// TwinCAT 3 PLC project TcOtel
// Title: TcOtel
// Company: AVM Engineering
// Author: Pirmin Bleiker
// ProjectVersion: 0.0.1
// ProgramVersion: 3.1.4026.22
// CompilerDefines: DEBUG
// libraries:
//   Tc2_EtherCAT, * (Beckhoff Automation GmbH)
//   Tc2_Standard, * (Beckhoff Automation GmbH)
//   Tc2_System, * (Beckhoff Automation GmbH)
//   Tc2_Utilities, * (Beckhoff Automation GmbH)
//   Tc3_Module, * (Beckhoff Automation GmbH)
//   TcUnit, * (www.tcunit.org)
//   Base Interfaces,newest,System
// project tree:
//   API/Context/ FB_ScopedContext.TcPOU, F_Context.TcPOU, I_ContextBuilder.TcIO
//   API/Log/ E_LogLevel.TcDUT, FB_Log.TcPOU (not stored), F_Log.TcPOU
//   API/Metric/ E_MetricStat.TcDUT, FB_Metrics.TcPOU
//   API/Trace/ FB_Trace.TcPOU (not stored), FB_Span.TcPOU (not stored), F_TraceParentFromString.TcPOU
//   API/Log/Interface/ I_LogBuilder.TcIO, I_WithLogger.TcIO, I_WithContext.TcIO, I_Logger.TcIO
//   API/ PRG_TaskLog.TcPOU (not stored)
//   DUTs/ E_CustomTypes.TcDUT, E_Scope.TcDUT, ST_TcOtelTaskInfo.TcDUT, ST_ScopedContextStack.TcDUT, E_TypeIdV2.TcDUT, ST_LogEntryHeaderV2.TcDUT, ST_SpanBeginPrefix.TcDUT, ST_SpanAttrFrame.TcDUT, ST_SpanEventFrame.TcDUT, ST_SpanEndFrame.TcDUT
//   GVLs/ Config.TcGVL (not stored), Const.TcGVL, TcOtelInfo.TcGVL
//   ITFs/ I_LogEntry.TcIO, I_LogEntryAdder.TcIO
//   POUs/Diagnostic/ FB_TcOtelTaskDiag.TcPOU, ST_PushDiagBatchHeader.TcDUT, ST_PushDiagConfig.TcDUT, ST_PushDiagSample.TcDUT
//   POUs/Logs/ FB_ContextBuilder.TcPOU, FB_LogBuilder.TcPOU, FB_LogEntry.TcPOU
//   POUs/Metrics/ E_MetricBodySchema.TcDUT, FB_TcOtelTaskMetrics.TcPOU, ST_DiagnosticCalculations.TcDUT, ST_PushMetricAggHeader.TcDUT
//   POUs/Trace/ E_SpanKind.TcDUT, E_SpanStatus.TcDUT, F_HashSpanId.TcPOU, F_HashTraceId.TcPOU, FB_TcOtelTaskTracer.TcPOU (not stored)
//   POUs/ FB_TcOtelTask.TcPOU (not stored), F_InternalLog.TcPOU (not stored), PRG_ScopedContextStack.TcPOU
//   POUs/Utils/ FB_LogBuffer.TcPOU, F_DINT_TO_UINT_MAX.TcPOU, IncUDINT.TcPOU
//   / ApiTest.TcPOU
//   Test/ FB_ContextBuilder_Test.TcPOU, PlcTask.TcTTO, PRG_Test.TcPOU
//   Version/ Global_Version.TcGVL
// real-time tasks:
//   TASK PlcTask: cycle T#1ms, priority 20, ADS port 350

CONFIGURATION TcOtel
    RESOURCE PLC ON TwinCAT3
        TASK PlcTask(INTERVAL := T#1ms, PRIORITY := 20);
        PROGRAM PRG_Test WITH PlcTask : PRG_Test;
    END_RESOURCE
END_CONFIGURATION

// ---- API/Log/E_LogLevel.TcDUT
(*
:Description: Definition of available log levels. 

The log levels are ordered. ``eTrace`` has the lowest priority, ``eFatal`` has the
highest priority.

===============
Log Level Usage
===============

Is is recommended to build a guidline for consistent use of the log level. A example
could be the following:

:eFatal: The fatal level should be used for any error which will to malfunction of the most
	part of the program. Log message of this type must be handled immedialtely.
	
	Example: A Safety controller could not be initialised

:eError: The error level should be used when the program cannot continue to work properly.
	Normally this means that a operator/user has to be alerted and something has to
	be fixed.

	Example: Communication errors, something stops a process

:eWarn: The warn level should be used when some expected condition has happend, but the
	software can proceed in some way or the operation can be repeated later. Normaly
	the warn level should be read by the user/operator at some time, not necessarly 
	immediately.

	Example: Cannot connect to some external system (but will repeat to try)

:eInfo: The info level should track some of the import state changes in the programm. This
	information can be used by the user/operator on demand to track a problem.

	Example: A state of a state-machine has changed, a new recipe has been loaded

:eDebug: The info level should track of the some internals, normally only of importance to
	developers.

:eTrace: The trace level should be used to track some internal processing. This is rarely
	used, even by developers, mostly to track some difficult problem.

*)
{attribute 'qualified_only'}
{attribute 'strict'}
{attribute 'to_string'}
TYPE E_LogLevel :
(
	eTrace 	:= 0,	(* Trace log level. *)
	eDebug 	:= 1,	(* Debug log level. *)
	eInfo	:= 2,	(* Info log level. *)
	eWarn	:= 3,	(* Warn log level. *)
	eError	:= 4,	(* Error log level. *)
	eFatal	:= 5,	(* Fatal log level. *)
	eDisabled := 99	(* Disabled *)
) UINT;
END_TYPE

// ---- API/Metric/E_MetricStat.TcDUT
(*
:Description: Bitmask values for the FB_Metrics aggregation stats.

Each bit selects one statistic that will be computed online (Welford
algorithm for mean / variance) over each sample interval and shipped as
8 bytes inside the body of an FB_Metrics aggregate frame
(``body_schema = eNumericAggregated``).

The wire-side ``nStatMask`` byte at header offset +0x11 is the OR of
the selected values. Body sample size = ``popcount(mask) * 8``. Stats
are written into the body in **bit-index order** (Min first if set,
then Max, then Mean, then Sum, then Count, then StdDev) — the decoder
walks the mask bit-by-bit and reads 8 bytes per set bit.

OR the values together to pick the stats you want:

.. code-block:: pascal

    fb.SetAggregation(E_MetricStat.eSum);                                   // counter
    fb.SetAggregation(E_MetricStat.eMin OR E_MetricStat.eMax);              // envelope
    fb.SetAggregation(E_MetricStat.eMin OR E_MetricStat.eMax
                      OR E_MetricStat.eMean);                               // recommended
    fb.SetAggregation(E_MetricStat.eMin OR E_MetricStat.eMax
                      OR E_MetricStat.eMean OR E_MetricStat.eSum
                      OR E_MetricStat.eCount OR E_MetricStat.eStdDev);      // full

Single-stat selections are valid and useful — e.g. ``eSum`` alone for
energy / counter metrics.
*)
TYPE E_MetricStat :
(
    eMin    := 16#01,    // bit 0
    eMax    := 16#02,    // bit 1
    eMean   := 16#04,    // bit 2 — Welford online mean
    eSum    := 16#08,    // bit 3 — total over the sample interval
    eCount  := 16#10,    // bit 4 — number of Observe() calls aggregated
    eStdDev := 16#20     // bit 5 — Welford online sample stddev
) BYTE;
END_TYPE

// ---- DUTs/E_CustomTypes.TcDUT
{attribute 'pack_mode' := '1'}
{attribute 'qualified_only'}
{attribute 'strict'}
TYPE INTERNAL E_CustomTypes :
(
	eType_TIME				:= 20000,
	eType_LTIME				:= 20001,
	eType_DATE				:= 20002,
	eType_DATE_AND_TIME		:= 20003,
	eType_TIME_OF_DAY		:= 20004,
	eType_ENUM				:= 20005,
	eType_WSTRING			:= 20006
) INT;
END_TYPE

// ---- DUTs/E_Scope.TcDUT
{attribute 'pack_mode' := '1'}
{attribute 'qualified_only'}
{attribute 'strict'}
{attribute 'conditionalshow'}
{attribute 'to_string'}
TYPE E_Scope :
(
	eLog			:= 0,
	eLogger			:= 1,
	eScoped			:= 2,
	eTask			:= 3
) BYTE;
END_TYPE

// ---- DUTs/ST_TcOtelTaskInfo.TcDUT
TYPE ST_TcOtelTaskInfo :
STRUCT
	nAddLogToBuffer						: UDINT;	(* Counts number of logs added to message buffer. *)
	nAddLogToBufferErrorCount			: UDINT;	(* Counts error when adding log message to task buffer. *)
	nSendLogBufferErrorCount			: UDINT;	(* Counts error when sending log task buffer to service. *)
	nMaxUsedBufferSize					: UDINT;	(* Max. used buffer size of log task buffer. *)
	bConnected							: BOOL;		(* TRUE when the service is reachable (last send succeeded). Logs are suppressed while FALSE. *)
	bReconnectPending					: BOOL;		(* TRUE on FALSE->TRUE bConnected edge; consumed by the task to emit a one-shot reconnect log. *)
END_STRUCT
END_TYPE

// ---- DUTs/ST_ScopedContextStack.TcDUT
{attribute 'conditionalshow'}
TYPE INTERNAL ST_ScopedContextStack :
STRUCT
	aScopedContext		: ARRAY[0..Config.nMaxScopedContext-1] OF I_ContextBuilder;
	nScopeContextCount	: UINT (0..Config.nMaxScopedContext);
END_STRUCT
END_TYPE

// ---- DUTs/E_TypeIdV2.TcDUT
{attribute 'pack_mode' := '1'}
{attribute 'qualified_only'}
{attribute 'strict'}
TYPE INTERNAL E_TypeIdV2 :
(
	eType_TIME_V2			:= 100,
	eType_LTIME_V2			:= 101,
	eType_DATE_V2			:= 102,
	eType_DATE_AND_TIME_V2	:= 103,
	eType_TIME_OF_DAY_V2	:= 104,
	eType_ENUM_V2			:= 105,
	eType_WSTRING_V2		:= 106
) BYTE;
END_TYPE

// ---- DUTs/ST_LogEntryHeaderV2.TcDUT
{attribute 'pack_mode' := '1'}
TYPE INTERNAL ST_LogEntryHeaderV2 :
STRUCT
	nType			: BYTE;		// 0x02 for v2 log entry
	nEntryLength	: UINT;		// Total length from after this field
	nLevel			: BYTE;		// Log level
	nTsPlc			: LINT;		// PLC timestamp (FILETIME)
	nTsClock		: LINT;		// Clock timestamp (FILETIME)
	nTaskIndex		: BYTE;		// Task index (0-63)
	nCycleCount		: UDINT;	// Cycle counter
	nArgCount		: BYTE;		// Argument count
	nContextCount	: BYTE;		// Context group count
END_STRUCT
END_TYPE

// ---- DUTs/ST_SpanBeginPrefix.TcDUT
(*
Fixed 24-byte prefix of a SPAN_BEGIN frame. Trace_id (16B) and span_id (8B)
follow immediately after, then the variable-length name and optional
external traceparent. Layout matches Rust parser_v2 BEGIN case.
*)
{attribute 'pack_mode' := '1'}
TYPE INTERNAL ST_SpanBeginPrefix :
STRUCT
    (* 12-byte common header *)
    nEventType      : BYTE;     (* 5 = SPAN_BEGIN *)
    nLocalId        : BYTE;     (* monotonic counter for SpanKey uniqueness *)
    nTaskIdx        : BYTE;
    nFlags          : BYTE;     (* bit1 = has_external_parent *)
    nDcTime         : LINT;     (* ns since DC epoch *)
    (* 12-byte begin meta *)
    abParentSpanId  : ARRAY[0..7] OF BYTE;
    nKind           : BYTE;
    nNameLen        : BYTE;
    nReserved       : ARRAY[0..1] OF BYTE;
END_STRUCT
END_TYPE

// ---- DUTs/ST_SpanAttrFrame.TcDUT
(*
Fixed 23-byte header of a SPAN_ATTR frame. Followed by key (nKeyLen bytes)
and value (nValueLen bytes). Layout matches Rust parser_v2 ATTR case.
*)
{attribute 'pack_mode' := '1'}
TYPE INTERNAL ST_SpanAttrFrame :
STRUCT
    (* 12-byte common header *)
    nEventType      : BYTE;     (* 6 = SPAN_ATTR *)
    nSpanIdByte0    : BYTE;     (* span_id[0] — shares slot with local_id *)
    nTaskIdx        : BYTE;
    nFlags          : BYTE;
    nDcTime         : LINT;
    (* 7-byte span_id rest *)
    abSpanIdRest    : ARRAY[0..6] OF BYTE;
    (* 4-byte attr meta *)
    nValueType      : BYTE;     (* 1=i64, 2=f64, 3=bool, 4=string *)
    nKeyLen         : BYTE;     (* ≤31 *)
    nValueLen       : BYTE;     (* wire bytes for value (1/8/N) *)
    nReserved       : BYTE;
END_STRUCT
END_TYPE

// ---- DUTs/ST_SpanEventFrame.TcDUT
(*
Fixed 23-byte header of a SPAN_EVENT frame. Followed by name (nNameLen bytes).
Layout matches Rust parser_v2 EVENT case.
*)
{attribute 'pack_mode' := '1'}
TYPE INTERNAL ST_SpanEventFrame :
STRUCT
    nEventType      : BYTE;     (* 7 = SPAN_EVENT *)
    nSpanIdByte0    : BYTE;
    nTaskIdx        : BYTE;
    nFlags          : BYTE;
    nDcTime         : LINT;
    abSpanIdRest    : ARRAY[0..6] OF BYTE;
    nNameLen        : BYTE;     (* ≤31 *)
    nAttrCount      : BYTE;     (* always 0 — inline attrs unused *)
    nReserved       : ARRAY[0..1] OF BYTE;
END_STRUCT
END_TYPE

// ---- DUTs/ST_SpanEndFrame.TcDUT
(*
Fixed 23-byte SPAN_END frame — no variable payload.
Layout matches Rust parser_v2 END case.
*)
{attribute 'pack_mode' := '1'}
TYPE INTERNAL ST_SpanEndFrame :
STRUCT
    nEventType      : BYTE;     (* 8 = SPAN_END *)
    nSpanIdByte0    : BYTE;
    nTaskIdx        : BYTE;
    nFlags          : BYTE;
    nDcTime         : LINT;
    abSpanIdRest    : ARRAY[0..6] OF BYTE;
    nStatus         : BYTE;     (* 1 = ok, 2 = error *)
    nMsgLen         : BYTE;     (* 0 — status_msg unused on wire today *)
    nReserved       : ARRAY[0..1] OF BYTE;
END_STRUCT
END_TYPE

// ---- POUs/Diagnostic/ST_PushDiagBatchHeader.TcDUT
(*
:Description: 80-byte header of a per-task diagnostic batch frame.

Prepended to an array of ``ST_PushDiagSample`` entries before pushing via
``ADSWRITE`` to tc-otel (IG = 16#4D424301, IO = 0). Packed tight
(``pack_mode := 1``) so on-wire layout matches the decoder in tc-otel-ads.
*)
  {attribute 'pack_mode' := '1'}
TYPE INTERNAL ST_PushDiagBatchHeader :
STRUCT
  version            : BYTE;                        // +0x00, wire version = 2
  event_type         : BYTE;                        // +0x01, event_type = 10 (batch)
  reserved0          : UINT;                        // +0x02, reserved = 0
  task_obj_id        : UDINT;                       // +0x04, TwinCAT task object id
  task_port          : UINT;                        // +0x08, AMS port of the owning task
  window_ms          : UINT;                        // +0x0A, aggregation window used for this batch (ms)
  sample_count       : UINT;                        // +0x0C, number of ST_PushDiagSample entries following
  reserved1          : UINT;                        // +0x0E, reserved = 0
  cycle_count_start  : UDINT;                       // +0x10, task cycle counter at first sample
  cycle_count_end    : UDINT;                       // +0x14, task cycle counter at last sample
  dc_time_start      : LINT;                        // +0x18, DC time at first sample (ns)
  dc_time_end        : LINT;                        // +0x20, DC time at last sample (ns)
  exec_time_min_us   : UDINT;                       // +0x28, min exec time in window (us)
  exec_time_max_us   : UDINT;                       // +0x2C, max exec time in window (us)
  exec_time_avg_us   : UDINT;                       // +0x30, avg exec time in window (us)
  cycle_exceed_count : UDINT;                       // +0x34, exceed cycles in window
  rt_violation_count : UDINT;                       // +0x38, rt-violation cycles in window
  task_name          : ARRAY [0..19] OF BYTE;       // +0x3C, task name (null-padded)
END_STRUCT
END_TYPE

// ---- POUs/Diagnostic/ST_PushDiagConfig.TcDUT
(*
:Description: Per-task push-diagnostic configuration, writable from tc-otel.

One instance per task lives in ``PRG_TaskLog.aTaskDiagConfig``. tc-otel can
update these slots at runtime via ADS SymbolByName writes so operators can
tune the aggregation window or disable push diagnostics from the UI without
recompiling the PLC project.

``divider = 0`` or ``divider = 1`` samples every cycle; ``divider = N`` keeps
every N-th cycle (useful on sub-100 us tasks where 1024 samples would fill
the ring too quickly).
*)
{attribute 'pack_mode' := '1'}
TYPE INTERNAL ST_PushDiagConfig :
STRUCT
  window_ms : UDINT := 100;           // +0x00, aggregation window in ms (flush interval)
  enabled   : BOOL := TRUE;            // +0x04, TRUE = collect and push samples
  divider   : USINT := 1;           // +0x05, 0/1 = every cycle, N = every N-th
  reserved  : UINT := 0;            // +0x06, reserved = 0, pad to 8 bytes
END_STRUCT
END_TYPE

// ---- POUs/Diagnostic/ST_PushDiagSample.TcDUT
(*
:Description: Single per-cycle diagnostic sample inside a push batch.

One sample is captured per PLC cycle and buffered in a 1024-entry ring inside
``FB_TcOtelTaskDiag``. The whole ring is flushed at the end of every
aggregation window. ``flags`` carries per-cycle markers:

* bit0 : cycle-time exceeded on this cycle
* bit1 : rt-violation on this cycle
* bit2 : first cycle after task start
* bit3 : ring buffer overflowed before this sample (samples lost)

Each sample keeps ``cycle_count`` and ``dc_time`` so tc-otel can correlate
flagged cycles back to the log entry produced on the same cycle.
*)
{attribute 'pack_mode' := '1'}
TYPE INTERNAL ST_PushDiagSample :
STRUCT
  cycle_count   : UDINT;                    // +0x00, task cycle counter
  exec_time_us  : UDINT;                    // +0x04, cycle execution time (us)
  dc_time       : LINT;                     // +0x08, distributed-clock time (ns)
  flags         : BYTE;                     // +0x10, per-cycle flag bits
  reserved      : ARRAY [0..6] OF BYTE;     // +0x11, padding to 24 bytes
END_STRUCT
END_TYPE

// ---- POUs/Metrics/E_MetricBodySchema.TcDUT
(*
:Description: Wire-format body schema for FB_Metrics push frames.

Encoded as a single byte at offset +0x03 of ST_PushMetricAggHeader. The
body of the frame is always sample_count * sample_size bytes; this enum
tells the receiver how to interpret each fixed-size slot.

Mapped from the locked IEC type at the first Observe() call. Numerics
(SINT..LREAL incl. unsigned) collapse to ``eNumeric`` and are widened
to LREAL (sample_size = 8). BOOL / discrete / strings keep their raw
sample size.
*)
TYPE INTERNAL E_MetricBodySchema :
(
    eUnknown            := 0,
    eBool               := 1,    // body: sample_count * 1 byte
    eNumeric            := 2,    // body: sample_count * 8 bytes (LREAL, widened)
    eDiscrete           := 3,    // body: sample_count * sample_size raw bytes (BYTE/WORD/DWORD/LWORD/ENUM)
    eString             := 4,    // body: sample_count * sample_size UTF-8 bytes (zero-padded fixed)
    eWstring            := 5,    // body: sample_count * sample_size UTF-16LE bytes (zero-padded fixed)
    eNumericAggregated  := 6     // body: sample_count * popcount(stat_mask) LREALs in bit-order
                                 // — see E_MetricStat for the bit assignments
) BYTE;
END_TYPE

// ---- POUs/Metrics/ST_DiagnosticCalculations.TcDUT
TYPE ST_DiagnosticCalculations :
STRUCT
	Count		: UDINT;
	Mean		: FLOAT;
	Minimum		: FLOAT;
	Maximum		: FLOAT;
	First		: FLOAT;
	Last		: FLOAT;
	Sum			: FLOAT;
	Variance	: FLOAT;
	Step		: FLOAT;
	Range		: FLOAT;
	StdDev		: FLOAT;
	Difference	: FLOAT;
END_STRUCT
END_TYPE

// ---- POUs/Metrics/ST_PushMetricAggHeader.TcDUT
(*
:Description: 52-byte fixed header of an FB_Metrics push frame.

The ``{attribute 'pack_mode' := '1'}`` pragma must be on the line **above
the TYPE keyword** (not inside the STRUCT body) — applied inside the
struct it would only act as a per-field hint and TwinCAT would still pad
the struct's tail to 8 bytes for the LINT members.

Pushed via ADSWRITE to ``IG = 0x4D424301`` / ``IO = 2`` (IO_PUSH_METRIC_AGG).
``event_type = 21`` (PUSH_METRIC_AGG) discriminates this frame from the
existing per-task diagnostic batch (event_type=10) and UI-driven custom
metric batch (event_type=20).

Wire layout (LE, ``pack_mode := 1``):

* +0x00 ``version``       — wire version = 2
* +0x01 ``event_type``    — = 21 (PUSH_METRIC_AGG)
* +0x02 ``flags``         — bit0=has_trace_ctx, bit1=ring_overflowed,
                             bit2=has_sample_ts
* +0x03 ``body_schema``   — see ``E_MetricBodySchema``
* +0x04 ``sample_size``   — bytes per sample in body
* +0x08 ``sample_count``  — number of samples in body
* +0x0C ``metric_id``     — FNV-1a hash of metric name (stable per name)
* +0x10 ``task_index``    — owning PLC task index (1..n)
* +0x11 ``stat_mask``     — bitmask of stats packed in body samples when
                            ``body_schema = eNumericAggregated`` (see
                            ``E_MetricStat``); 0 for raw / non-aggregated frames
* +0x12 reserved (2 B)    — pad to 4-byte alignment
* +0x14 ``cycle_count_start`` — task cycle counter at first sample in window
* +0x18 ``cycle_count_end``   — task cycle counter at last sample in window
* +0x1C reserved (4 B)        — pad to 8-byte alignment for ``dc_time_start``
* +0x20 ``dc_time_start``     — DC time at first sample (ns since DC epoch)
* +0x28 ``dc_time_end``       — DC time at last sample (ns since DC epoch)
* +0x30 ``name_len``          — bytes of metric name following the optional
                                 trace context (UTF-8, max 63)
* +0x31 ``unit_len``          — bytes of metric unit following ``name`` (UTF-8,
                                 max 15, 0 = unitless)
* +0x32 reserved (2 B)        — pad to 52 bytes
* = 0x34 (52 B) total fixed header

After this fixed header the frame contains, in order:

1. *Optional* — when ``flags.bit0 = 1`` — 24 B: trace_id (16 B) + span_id (8 B).
2. ``name_len`` bytes of metric name (UTF-8, no NUL).
3. ``unit_len`` bytes of metric unit (UTF-8, no NUL).
4. Body: ``sample_count`` sample slots. Slot layout depends on
   ``flags.bit2`` (has_sample_ts):

   * ``bit2 = 0`` (default): slot = ``sample_size`` value bytes. Total body
     = ``sample_count * sample_size``. Per-sample timestamps are reconstructed
     on the receiver side by linear interpolation between ``dc_time_start``
     and ``dc_time_end``.
   * ``bit2 = 1``: slot = 2 B ``cycle_offset`` (little-endian ``u16``,
     relative to ``cycle_count_start``) followed by ``sample_size`` value
     bytes. Total body = ``sample_count * (2 + sample_size)``. The receiver
     reconstructs per-sample DC time as
     ``dc_time_start + cycle_offset * cycle_time_ns`` where
     ``cycle_time_ns`` is derived from the header span. u16 covers up to
     65 535 cycles per window — the PLC emits an early autoflush if the
     configured push interval would exceed this.

Total frame size = 52 + (24 if has_trace_ctx else 0) + name_len + unit_len
                 + sample_count * (sample_size + (2 if has_sample_ts else 0)).
*)
{attribute 'pack_mode' := '1'}
TYPE ST_PushMetricAggHeader :
STRUCT
    nVersion           : BYTE;                      // +0x00, = 2
    nEventType         : BYTE;                      // +0x01, = 21
    nFlags             : BYTE;                      // +0x02, bit0=has_trace_ctx, bit1=ring_overflowed
    eBodySchema        : E_MetricBodySchema;        // +0x03, body interpretation tag
    nSampleSize        : UDINT;                     // +0x04, bytes per sample in body
    nSampleCount       : UDINT;                     // +0x08, samples in body
    nMetricId          : UDINT;                     // +0x0C, FNV-1a(name)
    nTaskIndex         : USINT;                     // +0x10, owning task index
    nStatMask          : BYTE;                      // +0x11, E_MetricStat bitmask (0 = raw/non-aggregated)
    aReserved0         : ARRAY [0..1] OF BYTE;      // +0x12, pad to 0x14
    nCycleCountStart   : UDINT;                     // +0x14
    nCycleCountEnd     : UDINT;                     // +0x18
    nReserved1         : UDINT;                     // +0x1C, pad to 0x20
    nDcTimeStart       : LINT;                      // +0x20
    nDcTimeEnd         : LINT;                      // +0x28
    nNameLen           : BYTE;                      // +0x30, max 63
    nUnitLen           : BYTE;                      // +0x31, max 15
    aReserved2         : ARRAY [0..1] OF BYTE;      // +0x32, pad to 52 bytes
END_STRUCT
END_TYPE

// ---- POUs/Trace/E_SpanKind.TcDUT
(*
:Description: Span kind enumeration for OpenTelemetry trace semantics.
*)
TYPE E_SpanKind :
(
    eInternal := 0,   (* Non-remote, internal-to-task operation *)
    eServer   := 1,   (* Handling an inbound RPC / request *)
    eClient   := 2,   (* Making an outbound RPC / request *)
    eProducer := 3,   (* Enqueueing onto an async queue / bus *)
    eConsumer := 4    (* Dequeueing from an async queue / bus *)
) USINT;
END_TYPE

// ---- POUs/Trace/E_SpanStatus.TcDUT
(*
:Description: Span completion status for OpenTelemetry traces.
*)
TYPE E_SpanStatus :
(
    eUnset := 0,  (* Unset status *)
    eOk    := 1,  (* Operation succeeded *)
    eError := 2   (* Operation failed *)
) USINT;
END_TYPE

// ---- GVLs/Const.TcGVL
{attribute 'qualified_only'}
VAR_GLOBAL CONSTANT
	sGlobalLogger		: STRING := '_GLOBAL_';		(* Global logger name for logger without logger input *)
	sLoggerFromInstance	: STRING := '__INST__';		(* FB_Logger*: Initialize logger name from instance path. *)
END_VAR

// ---- GVLs/TcOtelInfo.TcGVL
{attribute 'qualified_only'}
VAR_GLOBAL
	aTaskInfo							: ARRAY[1..SIZEOF(TwinCAT_SystemInfoVarList._TaskInfo)/SIZEOF(PlcTaskSystemInfo)] OF ST_TcOtelTaskInfo;
END_VAR

// ---- Version/Global_Version.TcGVL
{attribute 'TcGenerated'}
{attribute 'no-analysis'}
{attribute 'linkalways'}
// This function has been automatically generated from the project information.
VAR_GLOBAL CONSTANT
	{attribute 'const_non_replaced'}
	stLibVersion_TcOtel : ST_LibVersion := (iMajor := 0, iMinor := 0, iBuild := 1, iRevision := 0, nFlags := 0, sVersion := '0.0.1');
END_VAR

// ---- API/Context/I_ContextBuilder.TcIO
INTERFACE I_ContextBuilder EXTENDS __System.IQueryInterface

METHOD AddBool : I_ContextBuilder
VAR_INPUT
	sName		: T_MaxString;	
	bValue		: BOOL;
END_VAR
END_METHOD

METHOD AddByte : I_ContextBuilder
VAR_INPUT
	sName		: T_MaxString;
	nValue		: BYTE;
END_VAR
END_METHOD

METHOD AddDInt : I_ContextBuilder
VAR_INPUT
	sName		: T_MaxString;
	nValue		: DINT;
END_VAR
END_METHOD

METHOD AddDWord : I_ContextBuilder
VAR_INPUT
	sName	: Tc2_System.T_MaxString;
	nValue	: DWORD;
END_VAR
END_METHOD

METHOD AddInt : I_ContextBuilder
VAR_INPUT
	sName		: T_MaxString;
	nValue		: INT;
END_VAR
END_METHOD

METHOD AddLint : I_ContextBuilder
VAR_INPUT
	sName		: T_MaxString;
	nValue		: LINT;
END_VAR
END_METHOD

METHOD AddLReal : I_ContextBuilder
VAR_INPUT
	sName	: Tc2_System.T_MaxString;
	fValue	: LREAL;
END_VAR
END_METHOD

METHOD AddLWord : I_ContextBuilder
VAR_INPUT
	sName		: T_MaxString;
	nValue		: LWORD;
END_VAR
END_METHOD

METHOD AddReal : I_ContextBuilder
VAR_INPUT
	sName	: Tc2_System.T_MaxString;
	fValue	: REAL;
END_VAR
END_METHOD

METHOD AddSInt : I_ContextBuilder
VAR_INPUT
	sName		: T_MaxString;
	nValue		: SINT;
END_VAR
END_METHOD

METHOD AddString : I_ContextBuilder
VAR_INPUT
	sName		: T_MaxString;
	sValue		: T_MaxString;
END_VAR
END_METHOD

METHOD AddUDInt : I_ContextBuilder
VAR_INPUT
	sName		: T_MaxString;
	nValue		: UDINT;
END_VAR
END_METHOD

METHOD AddUInt : I_ContextBuilder
VAR_INPUT
	sName		: T_MaxString;
	nValue		: UINT;
END_VAR
END_METHOD

METHOD AddULint : I_ContextBuilder
VAR_INPUT
	sName		: T_MaxString;
	nValue		: ULINT;
END_VAR
END_METHOD

METHOD AddUSInt : I_ContextBuilder
VAR_INPUT
	sName		: T_MaxString;
	nValue		: USINT;
END_VAR
END_METHOD

METHOD AddWord : I_ContextBuilder
VAR_INPUT
	sName	: Tc2_System.T_MaxString;
	nValue	: WORD;
END_VAR
END_METHOD

METHOD Clear : I_ContextBuilder
VAR_INPUT
END_VAR
END_METHOD

METHOD Remove : I_ContextBuilder
VAR_INPUT
	sName	: Tc2_System.T_MaxString;
END_VAR
END_METHOD

END_INTERFACE

// ---- API/Log/Interface/I_LogBuilder.TcIO
// Fluent builder interface for composing log entries.
// Obtain an instance via F_Log() or FB_Log.Log(), chain methods, and call CreateLog() to emit.
INTERFACE I_LogBuilder EXTENDS I_WithContext, I_WithLogger

END_INTERFACE

// ---- API/Log/Interface/I_WithLogger.TcIO
// Fluent builder interface for composing log entries.
// Obtain an instance via F_Log() or FB_Log.Log(), chain methods, and call CreateLog() to emit.
INTERFACE I_WithLogger EXTENDS I_Logger

// Overrides the default logger name for this log entry.
// If not called, the global logger or FB_Log instance logger is used.
METHOD WithLogger : I_WithContext
VAR_INPUT
	sLogger	: T_MaxString;
END_VAR
END_METHOD

END_INTERFACE

// ---- API/Log/Interface/I_WithContext.TcIO
// Fluent builder interface for composing log entries.
// Obtain an instance via F_Log() or FB_Log.Log(), chain methods, and call CreateLog() to emit.
INTERFACE I_WithContext EXTENDS I_Logger

// Attaches context properties to this log entry.
// Use F_Context() to create a temporary context, or pass an FB_ContextBuilder instance.
METHOD WithContext : I_Logger
VAR_INPUT
	iContextBuilder	: I_ContextBuilder;
END_VAR
END_METHOD

(*
:Description: Bind this log entry to a specific FB_Span for explicit
trace context correlation.

When WithSpan is called, the log message will be associated with the span's
trace_id and span_id in the tc-otel backend, creating an explicit link in
the trace timeline.

Call before CreateLog to take effect. Calling after CreateLog has no effect.

Typical usage:

.. code-block:: pascal

    VAR
        spn : FB_Span;
    END_VAR

    F_Log(E_LogLevel.eInfo, 'operation started')
        .WithSpan(spn)
        .CreateLog();
*)
METHOD PUBLIC WithSpan : I_Logger
VAR_IN_OUT
	span : FB_Span;
END_VAR
END_METHOD

END_INTERFACE

// ---- API/Log/Interface/I_Logger.TcIO
// Fluent builder interface for composing log entries.
// Obtain an instance via F_Log() or FB_Log.Log(), chain methods, and call CreateLog() to emit.
INTERFACE I_Logger

// Finalizes and sends the log entry. Must be called to emit the log.
// After CreateLog(), the builder is consumed — do not reuse without a new F_Log() call.
METHOD CreateLog
END_METHOD

// Adds a log argument. Supports all IEC 61131-3 types (BOOL, INT, REAL, STRING, etc.).
// Arguments are referenced by position in the message template: '{0}', '{1}', ...
// Values are serialized immediately — safe to call in loops with changing variables.
METHOD WithAnyArg : I_Logger
VAR_INPUT
	stArg		: ANY;
END_VAR
END_METHOD

(*
:Description: Bind this log entry to a specific FB_Span for explicit
trace context correlation.

When WithSpan is called, the log message will be associated with the span's
trace_id and span_id in the tc-otel backend, creating an explicit link in
the trace timeline.

Call before CreateLog to take effect. Calling after CreateLog has no effect.

Typical usage:

.. code-block:: pascal

    VAR
        spn : FB_Span;
    END_VAR

    F_Log(E_LogLevel.eInfo, 'operation started')
        .WithSpan(spn)
        .CreateLog();
*)
METHOD PUBLIC WithSpan : I_Logger
VAR_IN_OUT
	span : FB_Span;
END_VAR
END_METHOD

// Adds a pre-typed argument (T_Arg from Tc2_Utilities).
// Prefer WithAnyArg for most cases. WithTArg is for compatibility with Tc2 formatting functions.
METHOD INTERNAL WithTArg : I_Logger
VAR_INPUT
	stArg		: T_Arg;
END_VAR
END_METHOD

END_INTERFACE

// ---- ITFs/I_LogEntry.TcIO
INTERFACE INTERNAL I_LogEntry EXTENDS __SYSTEM.IQueryInterface

METHOD PUBLIC AddAnyArg : BOOL
VAR_INPUT
	nArgNo		: BYTE;
	stArg		: ANY;
END_VAR
END_METHOD

METHOD INTERNAL AddBuffer
VAR_INPUT
	pBuffer			: PVOID;
	nBufferLen		: UDINT;
END_VAR
END_METHOD

METHOD PUBLIC AddContext
VAR_INPUT
	eScope			: E_Scope;
	pBuffer			: PVOID;
	nBufferLen		: UDINT;
END_VAR
END_METHOD

METHOD INTERNAL AddTArg
VAR_INPUT
	nArgNo		: BYTE;
	stArg		: Tc2_Utilities.T_Arg;
END_VAR
END_METHOD

METHOD PUBLIC End : BOOL
END_METHOD

METHOD INTERNAL Start : BOOL
VAR_INPUT
	pLogger		: POINTER TO T_MaxString;
	pMessage		: POINTER TO T_MaxString;
	eLogLevel		: E_LogLevel;
	nTimeStampPlc	: LINT;
	nTimeStampClock	: LINT;
END_VAR
END_METHOD

END_INTERFACE

// ---- ITFs/I_LogEntryAdder.TcIO
{attribute 'conditionalshow'}
INTERFACE INTERNAL I_LogEntryAdder EXTENDS __System.IQueryInterface

METHOD AddToLogEntry : BOOL
VAR_INPUT
	eScope			: E_Scope;
	iLogEntry		: I_LogEntry;
END_VAR
END_METHOD

END_INTERFACE

// ---- Test/PRG_Test.TcPOU
PROGRAM INTERNAL PRG_Test
VAR
	fbContextBuilder_Test	: FB_ContextBuilder_Test;

	fbLog			: FB_Log;

	fbScope			: FB_ScopedContext;
	bLog			: BOOL;
	bArg1			: BOOL;
	nArg2			: INT;
	sArg3			: STRING;


END_VAR

TcUnit.RUN();

IF _TaskInfo[GETCURTASKINDEXEX()].FirstCycle THEN
	// For Remote TC-OTel Server change the AMS net ID and configure a route
	PRG_TaskLog.Init('10.10.10.10.1.1');
	F_Log(E_LogLevel.eInfo, 'SPS Task gestartet.').CreateLog();
END_IF

fbLog.LoggerContext.AddInt('logger', 42);

IF bLog THEN
	bLog := FALSE;
	F_Log(E_LogLevel.eDebug, 'Foobar').CreateLog();
	F_Log(E_LogLevel.eInfo, '{0}, {1}, {2}')
		.WithAnyArg(bArg1)
		.WithAnyArg(nArg2)
		.WithAnyArg(sArg3)
		.CreateLog();

	fbLog.Info('barbaz {bLog}')
		.WithAnyArg(bLog)
		.CreateLog();
END_IF

PRG_TaskLog.Call();

END_PROGRAM

// ---- Test/FB_ContextBuilder_Test.TcPOU
FUNCTION_BLOCK INTERNAL FB_ContextBuilder_Test EXTENDS TcUnit.FB_TestSuite

AddInt_ShouldAddInt();
AddInt_WithSameName_ShouldReplace();
RemoveInt_ShouldRemove();

AddString_ShouldAddString();
AddString_WithSameName_ShouldReAdd();
AddString_WithSameName_ShouldReplace();
RemoveString_ShouldRemove();

METHOD AddInt_ShouldAddInt
VAR
	fbContextBuilder		: FB_ContextBuilder;
END_VAR
TcUnit.TEST('AddInt_ShouldAddInt');

fbContextBuilder.AddInt('foo', 42);

// 1 + 'foo' + 2 + 2
AssertEquals_UINT(8, fbContextBuilder._BufferCount, 'Buffer size');
AssertEquals_UINT(1, fbContextBuilder._ContextCount, 'Context count');
AssertEquals_UINT(0, fbContextBuilder._GetContextOffset(0), 'Context[0]');
AssertEquals_STRING('foo', fbContextBuilder._ReadName(0), 'Name');
AssertEquals_INT(Tc2_Utilities.E_ArgType.ARGTYPE_INT, fbContextBuilder._ReadType(0), 'Type');

TcUnit.TEST_FINISHED();
END_METHOD

METHOD AddInt_WithSameName_ShouldReplace
VAR
	fbContextBuilder		: FB_ContextBuilder;

END_VAR
TcUnit.TEST('AddInt_WithSameName_ShouldReplace');

// first add some
fbContextBuilder.AddInt('before', 0);	// size: 11
fbContextBuilder.AddWord('foo', 42);	// size: 8
fbContextBuilder.AddInt('after', 0);	// size: 10

// then replace
fbContextBuilder.AddInt('foo', 0);

AssertEquals_UINT(29, fbContextBuilder._BufferCount, 'Buffer size');
AssertEquals_UINT(3, fbContextBuilder._ContextCount, 'Context count');
AssertEquals_UINT(0, fbContextBuilder._GetContextOffset(0), 'Context[0]');
AssertEquals_UINT(11, fbContextBuilder._GetContextOffset(1), 'Context[1]');
AssertEquals_UINT(19, fbContextBuilder._GetContextOffset(2), 'Context[2]');
AssertEquals_STRING('before', fbContextBuilder._ReadName(0), 'Name[0]');
AssertEquals_STRING('foo', fbContextBuilder._ReadName(1), 'Name[1]');
AssertEquals_STRING('after', fbContextBuilder._ReadName(2), 'Name[2]');
AssertEquals_INT(Tc2_Utilities.E_ArgType.ARGTYPE_INT, fbContextBuilder._ReadType(1), 'Type');

TcUnit.TEST_FINISHED();
END_METHOD

METHOD AddString_ShouldAddString
VAR
	fbContextBuilder		: FB_ContextBuilder;
END_VAR
TcUnit.TEST('AddString_ShouldAddString');

fbContextBuilder.AddString('foo', 'bar');	// size: 10

AssertEquals_UINT(10, fbContextBuilder._BufferCount, 'Buffer size');
AssertEquals_UINT(1, fbContextBuilder._ContextCount, 'Context count');
AssertEquals_UINT(0, fbContextBuilder._GetContextOffset(0), 'Context[0]');
AssertEquals_STRING('foo', fbContextBuilder._ReadName(0), 'Name');
AssertEquals_INT(Tc2_Utilities.E_ArgType.ARGTYPE_STRING, fbContextBuilder._ReadType(0), 'Type');

TcUnit.TEST_FINISHED();
END_METHOD

METHOD AddString_WithSameName_ShouldReAdd
VAR
	fbContextBuilder		: FB_ContextBuilder;
END_VAR
TcUnit.TEST('AddString_WithSameName_ShouldReAdd');

fbContextBuilder.AddString('before', 'aaa');	// Size: 13
fbContextBuilder.AddString('foo', 'bar');		// Size: 10
fbContextBuilder.AddString('after', 'zzz');		// Size: 12

fbContextBuilder.AddString('foo', 'bazbar');	// Size: 13

AssertEquals_UINT(38, fbContextBuilder._BufferCount, 'Buffer size');
AssertEquals_UINT(3, fbContextBuilder._ContextCount, 'Context count');
AssertEquals_UINT(0, fbContextBuilder._GetContextOffset(0), 'Context[0]');
AssertEquals_UINT(13, fbContextBuilder._GetContextOffset(1), 'Context[1]');
AssertEquals_UINT(25, fbContextBuilder._GetContextOffset(2), 'Context[2]');
AssertEquals_STRING('before', fbContextBuilder._ReadName(0), 'Name[0]');
AssertEquals_STRING('after', fbContextBuilder._ReadName(1), 'Name[1]');
AssertEquals_STRING('foo', fbContextBuilder._ReadName(2), 'Name[2]');
AssertEquals_INT(Tc2_Utilities.E_ArgType.ARGTYPE_STRING, fbContextBuilder._ReadType(2), 'Type');

TcUnit.TEST_FINISHED();
END_METHOD

METHOD AddString_WithSameName_ShouldReplace
VAR
	fbContextBuilder		: FB_ContextBuilder;
END_VAR
TcUnit.TEST('AddString_WithSameName_ShouldReplace');

fbContextBuilder.AddString('before', 'aaa');	// Size: 13
fbContextBuilder.AddString('foo', 'bar');		// Size: 10
fbContextBuilder.AddString('after', 'zzz');		// Size: 12

fbContextBuilder.AddString('foo', 'baz');

AssertEquals_UINT(35, fbContextBuilder._BufferCount, 'Buffer size');
AssertEquals_UINT(3, fbContextBuilder._ContextCount, 'Context count');
AssertEquals_UINT(0, fbContextBuilder._GetContextOffset(0), 'Context[0]');
AssertEquals_UINT(13, fbContextBuilder._GetContextOffset(1), 'Context[1]');
AssertEquals_UINT(23, fbContextBuilder._GetContextOffset(2), 'Context[2]');
AssertEquals_STRING('before', fbContextBuilder._ReadName(0), 'Name[0]');
AssertEquals_STRING('foo', fbContextBuilder._ReadName(1), 'Name[1]');
AssertEquals_STRING('after', fbContextBuilder._ReadName(2), 'Name[2]');
AssertEquals_INT(Tc2_Utilities.E_ArgType.ARGTYPE_STRING, fbContextBuilder._ReadType(2), 'Type');

TcUnit.TEST_FINISHED();
END_METHOD

METHOD RemoveInt_ShouldRemove
VAR
	fbContextBuilder		: FB_ContextBuilder;

END_VAR
TcUnit.TEST('RemoveInt_ShouldRemove');

// first add some
fbContextBuilder.AddInt('before', 0);	// size: 11
fbContextBuilder.AddWord('foo', 42);	// size: 8
fbContextBuilder.AddInt('after', 0);	// size: 10

// then remove
fbContextBuilder.Remove('foo');

AssertEquals_UINT(21, fbContextBuilder._BufferCount, 'Buffer size');
AssertEquals_UINT(2, fbContextBuilder._ContextCount, 'Context count');
AssertEquals_UINT(0, fbContextBuilder._GetContextOffset(0), 'Context[0]');
AssertEquals_UINT(11, fbContextBuilder._GetContextOffset(1), 'Context[1]');
AssertEquals_STRING('before', fbContextBuilder._ReadName(0), 'Name[0]');
AssertEquals_STRING('after', fbContextBuilder._ReadName(1), 'Name[1]');

TcUnit.TEST_FINISHED();
END_METHOD

METHOD RemoveString_ShouldRemove
VAR
	fbContextBuilder		: FB_ContextBuilder;
END_VAR
TcUnit.TEST('RemoveString_ShouldRemove');

fbContextBuilder.AddString('before', 'aaa');	// Size: 13
fbContextBuilder.AddString('foo', 'bar');		// Size: 10
fbContextBuilder.AddString('after', 'zzz');		// Size: 12

fbContextBuilder.Remove('foo');

AssertEquals_UINT(25, fbContextBuilder._BufferCount, 'Buffer size');
AssertEquals_UINT(2, fbContextBuilder._ContextCount, 'Context count');
AssertEquals_UINT(0, fbContextBuilder._GetContextOffset(0), 'Context[0]');
AssertEquals_UINT(13, fbContextBuilder._GetContextOffset(1), 'Context[1]');
AssertEquals_STRING('before', fbContextBuilder._ReadName(0), 'Name[0]');
AssertEquals_STRING('after', fbContextBuilder._ReadName(1), 'Name[1]');

TcUnit.TEST_FINISHED();
END_METHOD

END_FUNCTION_BLOCK

// ---- POUs/Logs/FB_ContextBuilder.TcPOU
{attribute 'no_explicit_call' := 'no direct call necessary'}
{attribute 'conditionalshow'}
FUNCTION_BLOCK INTERNAL FB_ContextBuilder IMPLEMENTS I_ContextBuilder, I_LogEntryAdder
VAR CONSTANT
	nBufferSize			: UINT := 1024;
END_VAR
VAR
	aBuffer				: ARRAY[0..nBufferSize - 1] OF BYTE;	(* buffer for context variables *)
	nBufferCount		: UINT := 0;
	
	aContext			: ARRAY[0..19] OF UINT;
	nContextCount		: UINT(0..20) := 0;
END_VAR

METHOD PRIVATE _AddContext : BOOL
VAR_INPUT
	refName			: REFERENCE TO T_MaxString;
	nValueType		: INT;
	pValue			: PVOID;
	nValueLen		: UINT;
END_VAR
VAR
	nContextSize	: UINT;
	nNameLen		: INT;
	bOk				: BOOL;
END_VAR
_AddContext := FALSE;

IF nContextCount < 20 THEN
	nNameLen := Tc2_Standard.LEN(refName);
	IF nNameLen >= 0 AND nNameLen <= 255 THEN
		nContextSize :=
			INT_TO_UINT(nNameLen + 1) 		// String + Length-Byte
			+ INT_TO_UINT(SIZEOF(INT))		// Value type
			+ nValueLen;		// Value length

		IF (nBufferSize - nBufferCount) >= nContextSize  THEN
			aContext[nContextCount] := nBufferCount;
			nContextCount := nContextCount + 1;
		
			bOk :=
				_WriteByte(INT_TO_BYTE(nNameLen)) AND_THEN 
				_Copy(ADR(refName), INT_TO_UINT(nNameLen)) AND_THEN
				_WriteInt(nValueType) AND_THEN
				_Copy(pValue, nValueLen);
			
			IF bOk THEN
				_AddContext := TRUE;
			ELSE
				// Rollback
				nContextCount := nContextCount - 1;
				nBufferCount := aContext[nContextCount];
				
				F_InternalLog(
					E_LogLevel.eFatal,
					'FB_ContextBuilder._AddContext',
					'Error copy data to buffer - should not happen because of precheck',
					Tc2_Utilities.EMPTY_ARG_VALUE,
					Tc2_Utilities.EMPTY_ARG_VALUE,
					Tc2_Utilities.EMPTY_ARG_VALUE,
					Tc2_Utilities.EMPTY_ARG_VALUE
				);				
			END_IF
		ELSE
			F_InternalLog(
				E_LogLevel.eWarn,
				'FB_ContextBuilder._AddContext',
				'Too less space for adding context value %s.',
				Tc2_Utilities.F_StringEx(refName),
				Tc2_Utilities.EMPTY_ARG_VALUE,
				Tc2_Utilities.EMPTY_ARG_VALUE,
				Tc2_Utilities.EMPTY_ARG_VALUE
			);					
		END_IF
	ELSE
		// should not happen because T_MaxString is <= 255 bytes long
		F_InternalLog(
			E_LogLevel.eError,
			'FB_ContextBuilder._AddContext',
			'String longer than 255 bytes (actual=%d) - missin 0-byte?',
			Tc2_Utilities.F_INT(nNameLen),
			Tc2_Utilities.EMPTY_ARG_VALUE,
			Tc2_Utilities.EMPTY_ARG_VALUE,
			Tc2_Utilities.EMPTY_ARG_VALUE
		);		
	END_IF
ELSE
	F_InternalLog(
		E_LogLevel.eWarn,
		'FB_ContextBuilder._AddContext',
		'Number of context variable exceed (max. 20).',
		Tc2_Utilities.EMPTY_ARG_VALUE,
		Tc2_Utilities.EMPTY_ARG_VALUE,
		Tc2_Utilities.EMPTY_ARG_VALUE,
		Tc2_Utilities.EMPTY_ARG_VALUE
	);		
END_IF
END_METHOD

PROPERTY INTERNAL _BufferCount : UINT
GET
_BufferCount := nBufferCount;
END_GET
END_PROPERTY

PROPERTY INTERNAL _ContextCount : UINT
GET
_ContextCount := nContextCount;
END_GET
END_PROPERTY

METHOD PRIVATE _Copy : BOOL
VAR_INPUT
	pSrc		: PVOID;
	nCount		: UINT;
END_VAR
IF (nBufferSize - nBufferCount) >= nCount THEN
	MEMCPY(ADR(aBuffer) + nBufferCount, pSrc, nCount);
	nBufferCount := nBufferCount + nCount;
	
	_Copy := TRUE;
ELSE
	_Copy := FALSE;
END_IF
END_METHOD

METHOD PRIVATE _FindContext : UINT
VAR_INPUT
	refName		: REFERENCE TO Tc2_System.T_MaxString;
END_VAR
VAR
	nIdx		: UINT;
	nLen		: BYTE;
END_VAR
IF nContextCount > 0 THEN
	FOR nIdx := 0 TO nContextCount - 1 DO
		IF _ReadName(nIdx) = refName THEN
			_FindContext := nIdx;
			RETURN;
		END_IF
	END_FOR
END_IF

_FindContext := 16#FFFF;
END_METHOD

METHOD INTERNAL _GetContextOffset : UINT
VAR_INPUT
	nIdx		: UINT;
END_VAR
_GetContextOffset := aContext[nIdx];
END_METHOD

METHOD INTERNAL _GetDataLen : UINT
VAR_INPUT
	nIdx		: UINT;
END_VAR
VAR
	nSize		: UINT;
END_VAR
_GetDataLen := _GetSize(nIdx) - _GetOffsetToData(nIdx);
END_METHOD

METHOD PRIVATE _GetOffsetToData : UINT
VAR_INPUT
	nIdx		: UINT;
END_VAR
VAR
	pBuf		: PVOID;
	nOffset		: UINT;
END_VAR
pBuf := ADR(aBuffer) + aContext[nIdx];

// Offset to value (Skip name and type)
_GetOffsetToData := PBYTE_TO_BYTE(pBuf) + SIZEOF(BYTE) + SIZEOF(INT); // VARSTRING + INT
END_METHOD

METHOD PRIVATE _GetSize : UINT
VAR_INPUT
	nIdx		: UINT;
END_VAR
IF nIdx < nContextCount THEN
	IF (nIdx + 1) < nContextCount THEN
		_GetSize := aContext[nIdx + 1] - aContext[nIdx];
	ELSE
		_GetSize := nBufferCount - aContext[nIdx];
	END_IF
ELSE
	_GetSize := 0; 
END_IF
END_METHOD

METHOD INTERNAL _ReadName : T_MaxString
VAR_INPUT
	nIdx		: UINT;
END_VAR
VAR
	pBuf		: PVOID;
	nLen		: BYTE;
END_VAR
IF nIdx < nContextCount THEN
	pBuf := ADR(aBuffer) + aContext[nIdx];
	nLen := PBYTE_TO_BYTE(pBuf);
	MEMCPY(ADR(_ReadName), pBuf + 1, nLen);
	_ReadName[nLen] := 0;
ELSE
	_ReadName := '';	
END_IF
END_METHOD

METHOD INTERNAL _ReadType : INT
VAR_INPUT
	nIdx		: UINT;
END_VAR
VAR
	pBuf		: PVOID;
	nLen		: BYTE;
	nOffset		: UINT;
END_VAR
pBuf := ADR(aBuffer) + aContext[nIdx];

// Offset to value (Skip name and type)
nOffset := PBYTE_TO_BYTE(pBuf) + SIZEOF(BYTE); // VARSTRING + INT

MEMCPY(ADR(_ReadType), pBuf + nOffset, SIZEOF(INT));
END_METHOD

METHOD PRIVATE _RemoveContext : BOOL
VAR_INPUT
	refName		: REFERENCE TO Tc2_System.T_MaxString;
END_VAR
VAR
	nIdx		: UINT;
	nBufferOff	: UINT;
END_VAR
IF nContextCount > 0 THEN
	nIdx := _FindContext(refName);
	IF nIdx <> UINT#16#FFFF THEN
		(* Found - remove entry and compact buffer *)
		IF (nIdx + 1) < nContextCount THEN
			// Move buffer data
			MEMMOVE(
				ADR(aBuffer) + aContext[nIdx], 
				ADR(aBuffer) + aContext[nIdx + 1], 
				nBufferCount - aContext[nIdx + 1]
			);
			
			nBufferOff := aContext[nIdx + 1] - aContext[nIdx];
			nBufferCount := nBufferCount - nBufferOff;
			
			// Move and change index
			WHILE (nIdx + 1) < nContextCount DO
				aContext[nIdx] := aContext[nIdx + 1] - nBufferOff;
				nIdx := nIdx + 1;
			END_WHILE
		END_IF

		nContextCount := nContextCount - 1;
		_RemoveContext := TRUE;
		RETURN;
	END_IF
END_IF

_RemoveContext := FALSE;
END_METHOD

METHOD PRIVATE _ReplaceContext : BOOL
VAR_INPUT
	nIdx			: UINT;
	nValueType		: INT;
	pValue			: PVOID;
	nValueLen		: UINT;
END_VAR
VAR
	pBuf			: PVOID;
	nNameLen		: BYTE;
END_VAR
pBuf := ADR(aBuffer) + aContext[nIdx];

// Skip Name
nNameLen := PBYTE_TO_BYTE(pBuf);
pBuf := pBuf + nNameLen + 1;

pBuf := pBuf + MEMCPY(pBuf, ADR(nValueType), SIZEOF(nValueType));
pBuf := pBuf + MEMCPY(pBuf, pValue, nValueLen);
END_METHOD

METHOD PRIVATE _Reset
VAR_INPUT
END_VAR
nBufferCount := 0;
nContextCount := 0;
END_METHOD

METHOD PRIVATE _WriteByte : BOOL
VAR_INPUT
	nValue		: BYTE;
END_VAR
_WriteByte := _Copy(ADR(nValue), SIZEOF(nValue));
END_METHOD

METHOD PRIVATE _WriteInt : BOOL
VAR_INPUT
	nValue		: INT;
END_VAR
_WriteInt := _Copy(ADR(nValue), SIZEOF(nValue));
END_METHOD

METHOD AddBool : I_ContextBuilder
VAR_INPUT
	sName		: T_MaxString;
	bValue		: BOOL;
END_VAR
VAR
	nIdx	: UINT;
END_VAR
AddBool := THIS^;

nIdx := _FindContext(sName);
IF nIdx <> 16#FFFF THEN
	IF _GetDataLen(nIdx) = SIZEOF(bValue) THEN
		_ReplaceContext(nIdx, Tc2_Utilities.E_ArgType.ARGTYPE_BOOL, ADR(bValue), SIZEOF(bValue));
		RETURN;
	END_IF
	
	_RemoveContext(sName);
END_IF

_AddContext(
	refName		:= sName,
	nValueType	:= Tc2_Utilities.E_ArgType.ARGTYPE_BOOL,
	pValue		:= ADR(bValue),
	nValueLen	:= SIZEOF(bValue)
);
END_METHOD

METHOD AddByte : I_ContextBuilder
VAR_INPUT
	sName		: T_MaxString;
	nValue		: BYTE;
END_VAR
VAR
	nIdx	: UINT;
END_VAR
AddByte := THIS^;

nIdx := _FindContext(sName);
IF nIdx <> 16#FFFF THEN
	IF _GetDataLen(nIdx) = SIZEOF(nValue) THEN
		_ReplaceContext(nIdx, Tc2_Utilities.E_ArgType.ARGTYPE_BYTE, ADR(nValue), SIZEOF(nValue));
		RETURN;
	END_IF
	
	_RemoveContext(sName);
END_IF

_AddContext(
	refName		:= sName,
	nValueType	:= Tc2_Utilities.E_ArgType.ARGTYPE_BYTE,
	pValue		:= ADR(nValue),
	nValueLen	:= SIZEOF(nValue)
);
END_METHOD

METHOD AddDInt : I_ContextBuilder
VAR_INPUT
	sName	: Tc2_System.T_MaxString;
	nValue	: DINT;
END_VAR
VAR
	nIdx	: UINT;
END_VAR
AddDInt := THIS^;

nIdx := _FindContext(sName);
IF nIdx <> UINT#16#FFFF THEN
	IF _GetDataLen(nIdx) = SIZEOF(nValue) THEN
		_ReplaceContext(nIdx, Tc2_Utilities.E_ArgType.ARGTYPE_DINT, ADR(nValue), SIZEOF(nValue));
		RETURN;
	END_IF
	
	_RemoveContext(sName);
END_IF

_AddContext(
	refName		:= sName,
	nValueType	:= Tc2_Utilities.E_ArgType.ARGTYPE_DINT,
	pValue		:= ADR(nValue),
	nValueLen	:= SIZEOF(nValue)
);
END_METHOD

METHOD AddDWord : I_ContextBuilder
VAR_INPUT
	sName	: Tc2_System.T_MaxString;
	nValue	: DWORD;
END_VAR
VAR
	nIdx	: UINT;
END_VAR
AddDWord := THIS^;

nIdx := _FindContext(sName);
IF nIdx <> 16#FFFF THEN
	IF _GetDataLen(nIdx) = SIZEOF(nValue) THEN
		_ReplaceContext(nIdx, Tc2_Utilities.E_ArgType.ARGTYPE_DWORD, ADR(nValue), SIZEOF(nValue));
		RETURN;
	END_IF
	
	_RemoveContext(sName);
END_IF

_AddContext(
	refName		:= sName,
	nValueType	:= Tc2_Utilities.E_ArgType.ARGTYPE_DWORD,
	pValue		:= ADR(nValue),
	nValueLen	:= SIZEOF(nValue)
);
END_METHOD

METHOD AddInt : I_ContextBuilder
VAR_INPUT
	sName	: Tc2_System.T_MaxString;
	nValue	: INT;
END_VAR
VAR
	nIdx	: UINT;
END_VAR
AddInt := THIS^;

nIdx := _FindContext(sName);
IF nIdx <> UINT#16#FFFF THEN
	IF _GetDataLen(nIdx) = SIZEOF(nValue) THEN
		_ReplaceContext(nIdx, Tc2_Utilities.E_ArgType.ARGTYPE_INT, ADR(nValue), SIZEOF(nValue));
		RETURN;
	END_IF
	
	_RemoveContext(sName);
END_IF

_AddContext(
	refName		:= sName,
	nValueType	:= Tc2_Utilities.E_ArgType.ARGTYPE_INT,
	pValue		:= ADR(nValue),
	nValueLen	:= SIZEOF(nValue)
);
END_METHOD

METHOD AddLInt : I_ContextBuilder
VAR_INPUT
	sName	: Tc2_System.T_MaxString;
	nValue	: LINT;
END_VAR
VAR
	nIdx	: UINT;
END_VAR
AddLInt := THIS^;

nIdx := _FindContext(sName);
IF nIdx <> UINT#16#FFFF THEN
	IF _GetDataLen(nIdx) = SIZEOF(nValue) THEN
		_ReplaceContext(nIdx, Tc2_Utilities.E_ArgType.ARGTYPE_LARGE, ADR(nValue), SIZEOF(nValue));
		RETURN;
	END_IF
	
	_RemoveContext(sName);
END_IF

_AddContext(
	refName		:= sName,
	nValueType	:= Tc2_Utilities.E_ArgType.ARGTYPE_LARGE,
	pValue		:= ADR(nValue),
	nValueLen	:= SIZEOF(nValue)
);
END_METHOD

METHOD AddLReal : I_ContextBuilder
VAR_INPUT
	sName	: Tc2_System.T_MaxString;
	fValue	: LREAL;
END_VAR
VAR
	nIdx	: UINT;
END_VAR
AddLReal := THIS^;

nIdx := _FindContext(sName);
IF nIdx <> 16#FFFF THEN
	IF _GetDataLen(nIdx) = SIZEOF(fValue) THEN
		_ReplaceContext(nIdx, Tc2_Utilities.E_ArgType.ARGTYPE_LREAL, ADR(fValue), SIZEOF(fValue));
		RETURN;
	END_IF
	
	_RemoveContext(sName);
END_IF

_AddContext(
	refName		:= sName,
	nValueType	:= Tc2_Utilities.E_ArgType.ARGTYPE_LREAL,
	pValue		:= ADR(fValue),
	nValueLen	:= SIZEOF(fValue)
);
END_METHOD

METHOD AddLWord : I_ContextBuilder
VAR_INPUT
	sName	: Tc2_System.T_MaxString;
	nValue	: LWORD;
END_VAR
VAR
	nIdx	: UINT;
END_VAR
AddLWord := THIS^;

nIdx := _FindContext(sName);
IF nIdx <> UINT#16#FFFF THEN
	IF _GetDataLen(nIdx) = SIZEOF(nValue) THEN
		_ReplaceContext(nIdx, Tc2_Utilities.E_ArgType.ARGTYPE_LWORD, ADR(nValue), SIZEOF(nValue));
		RETURN;
	END_IF
	
	_RemoveContext(sName);
END_IF

_AddContext(
	refName		:= sName,
	nValueType	:= Tc2_Utilities.E_ArgType.ARGTYPE_LWORD,
	pValue		:= ADR(nValue),
	nValueLen	:= SIZEOF(nValue)
);
END_METHOD

METHOD AddReal : I_ContextBuilder
VAR_INPUT
	sName	: Tc2_System.T_MaxString;
	fValue	: REAL;
END_VAR
VAR
	nIdx	: UINT;
END_VAR
AddReal := THIS^;

nIdx := _FindContext(sName);
IF nIdx <> 16#FFFF THEN
	IF _GetDataLen(nIdx) = SIZEOF(fValue) THEN
		_ReplaceContext(nIdx, Tc2_Utilities.E_ArgType.ARGTYPE_REAL, ADR(fValue), SIZEOF(fValue));
		RETURN;
	END_IF
	
	_RemoveContext(sName);
END_IF

_AddContext(
	refName		:= sName,
	nValueType	:= Tc2_Utilities.E_ArgType.ARGTYPE_REAL,
	pValue		:= ADR(fValue),
	nValueLen	:= SIZEOF(fValue)
);
END_METHOD

METHOD AddSInt : I_ContextBuilder
VAR_INPUT
	sName	: Tc2_System.T_MaxString;
	nValue	: SINT;
END_VAR
VAR
	nIdx	: UINT;
END_VAR
AddSInt := THIS^;

nIdx := _FindContext(sName);
IF nIdx <> UINT#16#FFFF THEN
	IF _GetDataLen(nIdx) = SIZEOF(nValue) THEN
		_ReplaceContext(nIdx, Tc2_Utilities.E_ArgType.ARGTYPE_SINT, ADR(nValue), SIZEOF(nValue));
		RETURN;
	END_IF
	
	_RemoveContext(sName);
END_IF

_AddContext(
	refName		:= sName,
	nValueType	:= Tc2_Utilities.E_ArgType.ARGTYPE_SINT,
	pValue		:= ADR(nValue),
	nValueLen	:= SIZEOF(nValue)
);
END_METHOD

METHOD AddString : I_ContextBuilder
VAR_INPUT
	sName		: T_MaxString;
	sValue		: T_MaxString;
END_VAR
VAR
	nIdx		: UINT;
	aDataBuffer	: ARRAY[0..255] OF BYTE;
	nLen		: INT;
END_VAR
AddString := THIS^;

nLen := LEN(sValue);
IF nLen >= 0 AND nLen <= 255 THEN
	// copy string with length-byte into temporary buffer
	aDataBuffer[0] := INT_TO_BYTE(nLen);
	MEMCPY(ADR(aDataBuffer) + 1, ADR(sValue), INT_TO_UDINT(nLen));
	
	nIdx := _FindContext(sName);
	IF nIdx <> UINT#16#FFFF THEN
		IF _GetDataLen(nIdx) = INT_TO_UINT(nLen + 1) THEN
			_ReplaceContext(nIdx, Tc2_Utilities.E_ArgType.ARGTYPE_STRING, ADR(aDataBuffer), INT_TO_UINT(nLen) + 1);
			RETURN;
		END_IF
		
		_RemoveContext(sName);
	END_IF
	
	_AddContext(
		refName		:= sName,
		nValueType	:= E_ArgType.ARGTYPE_STRING,
		pValue		:= ADR(aDataBuffer),
		nValueLen	:= INT_TO_UINT(nLen) + 1
	);
ELSE
	F_InternalLog(
		E_LogLEvel.eFatal,
		'FB_ContextBuilder.AddString',
		'Pre check failed - string is longer than 255 (%d)',
		Tc2_Utilities.F_INT(nLen),
		Tc2_Utilities.EMPTY_ARG_VALUE,
		Tc2_Utilities.EMPTY_ARG_VALUE,
		Tc2_Utilities.EMPTY_ARG_VALUE
	);
END_IF
END_METHOD

METHOD AddToLogEntry : BOOL
VAR_INPUT
	eScope			: E_Scope;
	iLogEntry		: I_LogEntry;
END_VAR
VAR
	nIdx			: UINT;
	bOk				: BOOL;
	nContextLen		: UINT;
END_VAR
nIdx := 0;
bOk := TRUE;
IF iLogEntry = 0 THEN
	bOk := FALSE;
END_IF
WHILE nIdx < nContextCount AND bOk DO
	iLogEntry.AddContext(eScope, ADR(aBuffer) + aContext[nIdx], _GetSize(nIdx));
	nIdx := nIdx + 1;
END_WHILE

IF nIdx < nContextCount AND NOT bOk THEN
	F_InternalLog(
		E_LogLevel.eWarn,
		'FB_ContextBuilder.AddLogEntry',
		'Could not add all context properties to log entry. (act=%d, all=%d)',
		Tc2_Utilities.F_UINT(nIdx),
		Tc2_Utilities.F_UINT(nContextCount),
		Tc2_Utilities.EMPTY_ARG_VALUE,
		Tc2_Utilities.EMPTY_ARG_VALUE
	);
END_IF 

AddToLogEntry := bOk;
END_METHOD

METHOD AddUDInt : I_ContextBuilder
VAR_INPUT
	sName	: Tc2_System.T_MaxString;
	nValue	: UDINT;
END_VAR
VAR
	nIdx	: UINT;
END_VAR
AddUDInt := THIS^;

nIdx := _FindContext(sName);
IF nIdx <> UINT#16#FFFF THEN
	IF _GetDataLen(nIdx) = SIZEOF(nValue) THEN
		_ReplaceContext(nIdx, Tc2_Utilities.E_ArgType.ARGTYPE_UDINT, ADR(nValue), SIZEOF(nValue));
		RETURN;
	END_IF
	
	_RemoveContext(sName);
END_IF

_AddContext(
	refName		:= sName,
	nValueType	:= Tc2_Utilities.E_ArgType.ARGTYPE_UDINT,
	pValue		:= ADR(nValue),
	nValueLen	:= SIZEOF(nValue)
);
END_METHOD

METHOD AddUInt : I_ContextBuilder
VAR_INPUT
	sName	: Tc2_System.T_MaxString;
	nValue	: UINT;
END_VAR
VAR
	nIdx	: UINT;
END_VAR
AddUInt := THIS^;

nIdx := _FindContext(sName);
IF nIdx <> UINT#16#FFFF THEN
	IF _GetDataLen(nIdx) = SIZEOF(nValue) THEN
		_ReplaceContext(nIdx, Tc2_Utilities.E_ArgType.ARGTYPE_UINT, ADR(nValue), SIZEOF(nValue));
		RETURN;
	END_IF
	
	_RemoveContext(sName);
END_IF

_AddContext(
	refName		:= sName,
	nValueType	:= Tc2_Utilities.E_ArgType.ARGTYPE_UINT,
	pValue		:= ADR(nValue),
	nValueLen	:= SIZEOF(nValue)
);
END_METHOD

METHOD AddULInt : I_ContextBuilder
VAR_INPUT
	sName	: Tc2_System.T_MaxString;
	nValue	: ULINT;
END_VAR
VAR
	nIdx	: UINT;
END_VAR
AddULInt := THIS^;

nIdx := _FindContext(sName);
IF nIdx <> UINT#16#FFFF THEN
	IF _GetDataLen(nIdx) = SIZEOF(nValue) THEN
		_ReplaceContext(nIdx, Tc2_Utilities.E_ArgType.ARGTYPE_ULARGE, ADR(nValue), SIZEOF(nValue));
		RETURN;
	END_IF
	
	_RemoveContext(sName);
END_IF

_AddContext(
	refName		:= sName,
	nValueType	:= Tc2_Utilities.E_ArgType.ARGTYPE_ULARGE,
	pValue		:= ADR(nValue),
	nValueLen	:= SIZEOF(nValue)
);
END_METHOD

METHOD AddUSInt : I_ContextBuilder
VAR_INPUT
	sName	: Tc2_System.T_MaxString;
	nValue	: USINT;
END_VAR
VAR
	nIdx	: UINT;
END_VAR
AddUSInt := THIS^;

nIdx := _FindContext(sName);
IF nIdx <> UINT#16#FFFF THEN
	IF _GetDataLen(nIdx) = SIZEOF(nValue) THEN
		_ReplaceContext(nIdx, Tc2_Utilities.E_ArgType.ARGTYPE_USINT, ADR(nValue), SIZEOF(nValue));
		RETURN;
	END_IF
	
	_RemoveContext(sName);
END_IF

_AddContext(
	refName		:= sName,
	nValueType	:= Tc2_Utilities.E_ArgType.ARGTYPE_USINT,
	pValue		:= ADR(nValue),
	nValueLen	:= SIZEOF(nValue)
);
END_METHOD

METHOD AddWord : I_ContextBuilder
VAR_INPUT
	sName	: Tc2_System.T_MaxString;
	nValue	: WORD;
END_VAR
VAR
	nIdx	: UINT;
END_VAR
AddWord := THIS^;

nIdx := _FindContext(sName);
IF nIdx <> 16#FFFF THEN
	IF _GetDataLen(nIdx) = SIZEOF(nValue) THEN
		_ReplaceContext(nIdx, Tc2_Utilities.E_ArgType.ARGTYPE_WORD, ADR(nValue), SIZEOF(nValue));
		RETURN;
	END_IF
	
	_RemoveContext(sName);
END_IF

_AddContext(
	refName		:= sName,
	nValueType	:= Tc2_Utilities.E_ArgType.ARGTYPE_WORD,
	pValue		:= ADR(nValue),
	nValueLen	:= SIZEOF(nValue)
);
END_METHOD

METHOD Clear : I_ContextBuilder
VAR_INPUT
END_VAR
_Reset();
Clear := THIS^;
END_METHOD

METHOD Remove : I_ContextBuilder
VAR_INPUT
	sName	: Tc2_System.T_MaxString;
END_VAR
Remove := THIS^;
_RemoveContext(sName);
END_METHOD

END_FUNCTION_BLOCK

// ---- API/Context/FB_ScopedContext.TcPOU
(*
:Description: Provide nested scoped context properties. 

This function block can be used to define context properties, which
are valid from ``Begin()`` to ``End()``. This context properties can
be used to provide call-stack specific properties for example when
using multi-instance.

The maximum nested level can be configured with ``Config.nMaxScopedContext``.
The default level is 4.

**Example**

.. code:: 

	fbMachine1Ctx	: FB_ScopedContext;
	fbMachine2Ctx	: FB_ScopedContext;
	
	IF bInit THEN
		fbMachine1Ctx.ContextBuilder.AddInt('MachineNo', 1);
		fbMachine2Ctx.ContextBuilder.AddInt('MachineNo', 2);
	END_IF
	
    fbMachine1Ctx.Begin();
	// Call code for machine 1
	fbMachine1Ctx.End();
	
    fbMachine2Ctx.Begin();
	// Call code for machine 2
	fbMachine2Ctx.End();
*)
{attribute 'no_explicit_call' := 'no direct call necessary'}
FUNCTION_BLOCK PUBLIC FB_ScopedContext
VAR
	fbContext			: FB_ContextBuilder;
	bActive				: BOOL;
END_VAR

(*
:Description: Begins a nested context. 

Each ``Begin()`` call must be balance by an ``End()`` call in the same
order if nested context are used.
*)
METHOD PUBLIC Begin
VAR
	refTaskContextStack		: REFERENCE TO ST_ScopedContextStack;
END_VAR
IF NOT bActive THEN
	bActive := TRUE;
	
	refTaskContextStack REF= PRG_ScopedContextStack.TaskContextStack;
	
	IF refTaskContextStack.nScopeContextCount < Config.nMaxScopedContext THEN
		refTaskContextStack.aScopedContext[refTaskContextStack.nScopeContextCount] := fbContext;
		refTaskContextStack.nScopeContextCount := refTaskContextStack.nScopeContextCount + 1;
	ELSE
		F_InternalLog(
			E_LogLevel.eError,
			'FB_ScopedContext.Begin',
			'Too many nested scoped context.',
			Tc2_Utilities.EMPTY_ARG_VALUE,
			Tc2_Utilities.EMPTY_ARG_VALUE,
			Tc2_Utilities.EMPTY_ARG_VALUE,
			Tc2_Utilities.EMPTY_ARG_VALUE
		);
	END_IF
ELSE
	F_InternalLog(
		E_LogLevel.eError,
		'FB_ScopedContext.Begin',
		'Begin() called twice without End()',
		Tc2_Utilities.EMPTY_ARG_VALUE,
		Tc2_Utilities.EMPTY_ARG_VALUE,
		Tc2_Utilities.EMPTY_ARG_VALUE,
		Tc2_Utilities.EMPTY_ARG_VALUE
	);
END_IF
END_METHOD

(*
:Description: Returns the context builder for this scoped context. 

For best performance the context build should only be called on
changed values.
*)
PROPERTY PUBLIC ContextBuilder : I_ContextBuilder
GET
ContextBuilder := fbContext;
END_GET
END_PROPERTY

(*
:Description: Ends a nested context. 

Each ``Begin()`` call must be balance by an ``End()`` call in the same
order if nested context are used.
*)
METHOD PUBLIC End
VAR
	nIdx					: INT;
	refTaskContextStack		: REFERENCE TO ST_ScopedContextStack;
	iThisContextBuilder		: I_ContextBuilder;
END_VAR
IF bActive THEN
	bActive := FALSE;
	
	refTaskContextStack REF= PRG_ScopedContextStack.TaskContextStack;
	iThisContextBuilder := fbContext;
	
	// expected at top
	IF refTaskContextStack.nScopeContextCount > 0 
			AND_THEN refTaskContextStack.aScopedContext[refTaskContextStack.nScopeContextCount - 1] = iThisContextBuilder 
	THEN
		refTaskContextStack.nScopeContextCount := refTaskContextStack.nScopeContextCount - 1;
		RETURN;
	END_IF
	
	// try to find it in the stack
	FOR nIdx := UINT_TO_INT(refTaskContextStack.nScopeContextCount) - 1 TO 0 BY -1 DO
		IF refTaskContextStack.aScopedContext[nIdx] = iThisContextBuilder THEN
			F_InternalLog(
				E_LogLevel.eError,
				'FB_ScopedContext.End',
				'Removed scoped context at %d instead of %d-1 - ensure Begin/End are called in order.',
				Tc2_Utilities.F_INT(nIdx),
				Tc2_Utilities.F_UINT(refTaskContextStack.nScopeContextCount),
				Tc2_Utilities.EMPTY_ARG_VALUE,
				Tc2_Utilities.EMPTY_ARG_VALUE
			);	
		
			refTaskContextStack.nScopeContextCount := INT_TO_UINT(nIdx);
			RETURN;
		END_IF
	END_FOR
	
	F_InternalLog(
		E_LogLevel.eError,
		'FB_ScopedContext.End',
		'Cannot remove non existing scope',
		Tc2_Utilities.EMPTY_ARG_VALUE,
		Tc2_Utilities.EMPTY_ARG_VALUE,
		Tc2_Utilities.EMPTY_ARG_VALUE,
		Tc2_Utilities.EMPTY_ARG_VALUE
	);	
ELSE
	F_InternalLog(
		E_LogLevel.eError,
		'FB_ScopedContext.End',
		'End() called without Begin()',
		Tc2_Utilities.EMPTY_ARG_VALUE,
		Tc2_Utilities.EMPTY_ARG_VALUE,
		Tc2_Utilities.EMPTY_ARG_VALUE,
		Tc2_Utilities.EMPTY_ARG_VALUE
	);
END_IF
END_METHOD

END_FUNCTION_BLOCK

// ---- POUs/PRG_ScopedContextStack.TcPOU
{attribute 'conditionalshow'}
PROGRAM INTERNAL PRG_ScopedContextStack
VAR
	aContextStack		: ARRAY[1..SIZEOF(TwinCAT_SystemInfoVarList._TaskInfo)/SIZEOF(PlcTaskSystemInfo)] OF ST_ScopedContextStack;
END_VAR

PROPERTY INTERNAL TaskContextStack : REFERENCE TO ST_ScopedContextStack
GET
VAR
	nTaskIdx	: DINT;
END_VAR
nTaskIdx := Tc2_System.GETCURTASKINDEXEX();
TaskContextStack REF= aContextStack[nTaskIdx];
END_GET
END_PROPERTY

END_PROGRAM

// ---- API/Log/F_Log.TcPOU
FUNCTION F_Log : I_LogBuilder
VAR_INPUT
	eLogLevel		: E_LogLevel;
	sMessage		: T_MaxString;
END_VAR
VAR_STAT
	aLogBuilder		: ARRAY[1..SIZEOF(TwinCAT_SystemInfoVarList._TaskInfo)/SIZEOF(PlcTaskSystemInfo)] OF FB_LogBuilder;
END_VAR

F_Log := aLogBuilder[Tc2_System.GETCURTASKINDEXEX()].Clear(sMessage := sMessage, eLogLevel := eLogLevel);

END_FUNCTION

// ---- POUs/Logs/FB_LogBuilder.TcPOU
{attribute 'no_explicit_call' := 'no direct call necessary'}
{attribute 'conditionalshow'}
FUNCTION_BLOCK INTERNAL FB_LogBuilder IMPLEMENTS I_LogBuilder
VAR
	sMessage			: T_MaxString;
	eLogLevel			: E_LogLevel;
	sLogger				: T_MaxString := Const.sGlobalLogger;
	fbLogEntry			: FB_LogEntry();
	iLogEntryAdder		: I_LogEntryAdder;
	nIdx				: UINT;
	refScopedContext	: REFERENCE TO ST_ScopedContextStack;
	iContextBuilder		: I_ContextBuilder;
	bStarted			: BOOL;		// TRUE after StartV2 has been called
	bError				: BOOL;
	(* Phase 6 Stage 4: span reference for explicit log-to-trace correlation.
	   Set via WithSpan for logs that should be correlated to a specific span.
	   NULL (default) means no span correlation. *)
	_pSpan				: REFERENCE TO FB_Span;
END_VAR

METHOD PRIVATE _EnsureStarted
IF bStarted OR bError THEN
	RETURN;
END_IF

fbLogEntry.StartV2(
	pLogger			:= ADR(THIS^.sLogger),
	pMessage		:= ADR(THIS^.sMessage),
	eLogLevel		:= eLogLevel,
	nTimeStampPlc	:= 0,
	nTimeStampClock	:= 0
);
bStarted := TRUE;
END_METHOD

METHOD PRIVATE _IsLogLevelActive : BOOL
VAR_INPUT
END_VAR
// Suppress both when the log level is below the configured threshold AND when
// the service is not reachable. Skipping unreachable logs avoids all downstream
// MEMCPY work (message, logger name, args, context) while disconnected.
_IsLogLevelActive := eLogLevel >= Config.eMaxLogLevel
	AND TcOtelInfo.aTaskInfo[Tc2_System.GETCURTASKINDEXEX()].bConnected;
END_METHOD

METHOD INTERNAL Clear : I_LogBuilder
VAR_IN_OUT
	sMessage		: T_MaxString;
END_VAR
VAR_INPUT
	eLogLevel		: E_LogLevel;
	pLogger			: POINTER TO T_MaxString := 0;
END_VAR
Clear := THIS^;
THIS^.eLogLevel := eLogLevel;
IF NOT _IsLogLevelActive() THEN
	RETURN;
END_IF
THIS^.fbLogEntry.Reset();
THIS^.iContextBuilder := 0;
THIS^._pSpan REF= 0;
THIS^.sMessage := sMessage;
IF pLogger <> 0 THEN
	THIS^.sLogger := pLogger^;
ELSE
	THIS^.sLogger := Const.sGlobalLogger;
END_IF
bStarted := FALSE;
bError := FALSE;
END_METHOD

METHOD CreateLog
IF NOT _IsLogLevelActive() THEN
	RETURN;
END_IF

// Ensure header+message+logger are written (in case no args were added)
_EnsureStarted();

// Context comes after args in the wire format
IF __QUERYINTERFACE(PRG_TaskLog.TaskLogger.TaskContext, iLogEntryAdder) THEN
	iLogEntryAdder.AddToLogEntry(E_Scope.eTask, fbLogEntry);
END_IF

refScopedContext REF= PRG_ScopedContextStack.TaskContextStack;
IF refScopedContext.nScopeContextCount > 0 THEN
	FOR nIdx := 0 TO refScopedContext.nScopeContextCount - 1 DO
		IF __QUERYINTERFACE(refScopedContext.aScopedContext[nIdx], iLogEntryAdder) THEN
			iLogEntryAdder.AddToLogEntry(E_Scope.eScoped, fbLogEntry);
		END_IF
	END_FOR
END_IF

IF iContextBuilder <> 0 AND __QUERYINTERFACE(iContextBuilder, iLogEntryAdder) THEN
	iLogEntryAdder.AddToLogEntry(E_Scope.eLogger, fbLogEntry);
END_IF

fbLogEntry.End();
END_METHOD

METHOD WithAnyArg : I_Logger
VAR_INPUT
	stArg	: ANY;
END_VAR
WithAnyArg := THIS^;
IF NOT _IsLogLevelActive() THEN
	RETURN;
END_IF

// Lazy start: write header+message+logger on first arg
_EnsureStarted();

// Write arg directly into LogEntry buffer (v2 format)
fbLogEntry.AddAnyArg(0, stArg);
END_METHOD

METHOD WithContext : I_Logger
VAR_INPUT
	iContextBuilder	: I_ContextBuilder;
END_VAR
WithContext := THIS^;
IF NOT _IsLogLevelActive() THEN
	RETURN;
END_IF
THIS^.iContextBuilder := iContextBuilder;
END_METHOD

METHOD WithLogger : I_WithContext
VAR_INPUT
	sLogger	: T_MaxString;
END_VAR
WithLogger := THIS^;
IF NOT _IsLogLevelActive() THEN
	RETURN;
END_IF
THIS^.sLogger := sLogger;
END_METHOD

(*
:Description: Bind this log entry to a specific FB_Span for explicit
trace context correlation.

When WithSpan is called, the log message will be associated with the span's
trace_id and span_id in the tc-otel backend, creating an explicit link in
the trace timeline.

Call before CreateLog to take effect. Calling after CreateLog has no effect.

Typical usage:

.. code-block:: pascal

    VAR
        spn : FB_Span;
    END_VAR

    F_Log(E_LogLevel.eInfo, 'operation started')
        .WithSpan(spn)
        .CreateLog();
*)
METHOD PUBLIC WithSpan : I_Logger
VAR_IN_OUT
	span : FB_Span;
END_VAR
WithSpan := THIS^;
IF NOT _IsLogLevelActive() THEN
	RETURN;
END_IF

_pSpan REF= span;
END_METHOD

METHOD WithTArg : I_Logger
VAR_INPUT
	stArg	: T_Arg;
END_VAR
WithTArg := THIS^;
IF NOT _IsLogLevelActive() THEN
	RETURN;
END_IF

// Lazy start: write header+message+logger on first arg
_EnsureStarted();

// Write arg directly into LogEntry buffer
fbLogEntry.AddTArg(0, stArg);
END_METHOD

END_FUNCTION_BLOCK

// ---- POUs/Logs/FB_LogEntry.TcPOU
{attribute 'no_explicit_call' := 'no direct call necessary'} 
{attribute 'conditionalshow'}
FUNCTION_BLOCK INTERNAL FB_LogEntry IMPLEMENTS I_LogEntry
VAR
	pBuffer				: PVOID;	// pointer to the current message buffer
	nBufferCount		: UDINT;	// number of bytes written to the message buffer
	nBufferRemaining	: UDINT;	// remaining bytes in the message buffer
	bError				: BOOL;		// indicates an error in the current message building
	// v2 Protocol fields
	nEntryStart			: UDINT;	// Buffer position where entry begins
	nEntryLenOffset		: UDINT;	// Position of entry_length field (for backfill)
	nArgCountOffset		: UDINT;	// Position of arg_count field (for backfill)
	nCtxCountOffset		: UDINT;	// Position of context_count field (for backfill)
	nArgCount			: BYTE;		// Argument count (v2 only)
	nContextCount		: BYTE;		// Context group count (v2 only)
	bV2					: BOOL;		// TRUE if v2 protocol is active
END_VAR

METHOD PRIVATE _Copy
VAR_INPUT
	pSrc		: PVOID;
	nCount		: UDINT;
END_VAR
IF NOT bError AND_THEN nBufferRemaining >= nCount THEN
	Tc2_System.MEMCPY(pBuffer + nBufferCount, pSrc, nCount);
	nBufferCount := nBufferCount + nCount;
	nBufferRemaining := nBufferRemaining - nCount;
ELSE
	IF NOT bError THEN
		F_InternalLog(
			E_LogLevel.eWarn,
			'FB_LogEntry._Copy',
			'Error buffer overflow for log message (act=%d, new=%d)',
			Tc2_Utilities.F_UDINT(nBufferCount),
			Tc2_Utilities.F_UDINT(nCount),
			Tc2_Utilities.EMPTY_ARG_VALUE,
			Tc2_Utilities.EMPTY_ARG_VALUE
		);
	END_IF
	bError := TRUE;
END_IF
END_METHOD

METHOD PRIVATE _Reset
VAR
	pWriteBuffer	: REFERENCE TO FB_LogBuffer;
END_VAR
pWriteBuffer REF= PRG_TaskLog.TaskLogger.WriteBuffer;
pBuffer := pWriteBuffer.BufferPtr;
nBufferCount := 0;
nBufferRemaining := pWriteBuffer.BufferFree;

bError := FALSE;
END_METHOD

METHOD PRIVATE _WriteByte 
VAR_INPUT
	nValue		: BYTE;
END_VAR
_Copy(ADR(nValue), SIZEOF(nValue));
END_METHOD

METHOD PRIVATE _WriteDInt
VAR_INPUT
	nValue		: DINT;
END_VAR
_Copy(ADR(nValue), SIZEOF(nValue));
END_METHOD

METHOD PRIVATE _WriteInt 
VAR_INPUT
	nValue		: INT;
END_VAR
_Copy(ADR(nValue), SIZEOF(nValue));
END_METHOD

METHOD PRIVATE _WriteLInt
VAR_INPUT
	nValue		: LINT;
END_VAR
_Copy(ADR(nValue), SIZEOF(nValue));
END_METHOD

METHOD PRIVATE _WriteString
VAR_INPUT
	pValue		: POINTER TO Tc2_Utilities.T_MaxString;
END_VAR
VAR
	nLen			: INT;
END_VAR
IF pValue <> 0 THEN
	nLen := TO_INT(Tc2_Utilities.LEN2(pValue));
	IF nLen >= 0 AND nLen <= 255 THEN
		_WriteByte(INT_TO_BYTE(nLen)); 
		_Copy(pValue, INT_TO_UINT(nLen));
	ELSE
		// should not happen because T_MaxString is <= 255 bytes long
		bError := TRUE;
		F_InternalLog(
			E_LogLevel.eError,
			'FB_LogEntry._WriteString',
			'String longer than 255 bytes (actual=%d) - missin 0-byte?',
			Tc2_Utilities.F_INT(nLen),
			Tc2_Utilities.EMPTY_ARG_VALUE,
			Tc2_Utilities.EMPTY_ARG_VALUE,
			Tc2_Utilities.EMPTY_ARG_VALUE
		);
	END_IF
ELSE
		bError := TRUE;
		F_InternalLog(
			E_LogLevel.eError,
			'FB_LogEntry._WriteString',
			'String null pointer',
			Tc2_Utilities.EMPTY_ARG_VALUE,
			Tc2_Utilities.EMPTY_ARG_VALUE,
			Tc2_Utilities.EMPTY_ARG_VALUE,
			Tc2_Utilities.EMPTY_ARG_VALUE
		);
END_IF
END_METHOD

METHOD PRIVATE _WriteUDInt
VAR_INPUT
	nValue		: UDINT;
END_VAR
_Copy(ADR(nValue), SIZEOF(nValue));
END_METHOD

METHOD PRIVATE _WriteUInt 
VAR_INPUT
	nValue		: UINT;
END_VAR
_Copy(ADR(nValue), SIZEOF(nValue));
END_METHOD

METHOD PRIVATE _WriteULInt
VAR_INPUT
	nValue		: ULINT;
END_VAR
_Copy(ADR(nValue), SIZEOF(nValue));
END_METHOD

METHOD PRIVATE _WriteWString
VAR_INPUT
	pValue		: POINTER TO WSTRING(255);
END_VAR
VAR
	nLen			: INT;
END_VAR
IF pValue <> 0 THEN
	nLen := Tc2_Standard.WLEN(pValue^);
	IF nLen >= 0 AND nLen <= 255 THEN
		_WriteByte(INT_TO_BYTE(nLen)); 
		_Copy(pValue, INT_TO_UINT(nLen) * 2);
	ELSE
		// should not happen because T_MaxString is <= 255 bytes long
		bError := TRUE;
		F_InternalLog(
			E_LogLevel.eError,
			'FB_LogEntry._WriteWString',
			'String longer than 255 bytes (actual=%d) - missin 0-byte?',
			Tc2_Utilities.F_INT(nLen),
			Tc2_Utilities.EMPTY_ARG_VALUE,
			Tc2_Utilities.EMPTY_ARG_VALUE,
			Tc2_Utilities.EMPTY_ARG_VALUE
		);
	END_IF
ELSE
		bError := TRUE;
		F_InternalLog(
			E_LogLevel.eError,
			'FB_LogEntry._WriteWString',
			'String null pointer',
			Tc2_Utilities.EMPTY_ARG_VALUE,
			Tc2_Utilities.EMPTY_ARG_VALUE,
			Tc2_Utilities.EMPTY_ARG_VALUE,
			Tc2_Utilities.EMPTY_ARG_VALUE
		);
END_IF
END_METHOD

METHOD PUBLIC AddAnyArg : BOOL
VAR_INPUT
	nArgNo		: BYTE;
	stArg		: ANY;
END_VAR
VAR
	nLen		: INT;
END_VAR
IF bError THEN
	RETURN;
END_IF

IF stArg.pValue = 0 THEN
	RETURN;
END_IF

IF bV2 THEN
	// v2 format: type_id as 1 byte, no marker byte, no index byte
	CASE stArg.TypeClass OF
		__SYSTEM.TYPE_CLASS.TYPE_BOOL:
			_WriteByte(TO_BYTE(Tc2_Utilities.E_ArgType.ARGTYPE_BOOL));
			IF Tc2_Utilities.PBYTE_TO_BYTE(stArg.pValue) <> 0 THEN
				_WriteByte(1);
			ELSE
				_WriteByte(0);
			END_IF

		__SYSTEM.TYPE_CLASS.TYPE_BYTE:
			_WriteByte(TO_BYTE(Tc2_Utilities.E_ArgType.ARGTYPE_BYTE));
			_Copy(stArg.pValue, SIZEOF(BYTE));

		__SYSTEM.TYPE_CLASS.TYPE_WORD:
			_WriteByte(TO_BYTE(Tc2_Utilities.E_ArgType.ARGTYPE_WORD));
			_Copy(stArg.pValue, SIZEOF(WORD));

		__SYSTEM.TYPE_CLASS.TYPE_DWORD:
			_WriteByte(TO_BYTE(Tc2_Utilities.E_ArgType.ARGTYPE_DWORD));
			_Copy(stArg.pValue, SIZEOF(DWORD));

		__SYSTEM.TYPE_CLASS.TYPE_LWORD:
			_WriteByte(TO_BYTE(Tc2_Utilities.E_ArgType.ARGTYPE_LWORD));
			_Copy(stArg.pValue, SIZEOF(LWORD));

		__SYSTEM.TYPE_CLASS.TYPE_SINT:
			_WriteByte(TO_BYTE(Tc2_Utilities.E_ArgType.ARGTYPE_SINT));
			_Copy(stArg.pValue, SIZEOF(SINT));

		__SYSTEM.TYPE_CLASS.TYPE_INT:
			_WriteByte(TO_BYTE(Tc2_Utilities.E_ArgType.ARGTYPE_INT));
			_Copy(stArg.pValue, SIZEOF(INT));

		__SYSTEM.TYPE_CLASS.TYPE_DINT:
			_WriteByte(TO_BYTE(Tc2_Utilities.E_ArgType.ARGTYPE_DINT));
			_Copy(stArg.pValue, SIZEOF(DINT));

		__SYSTEM.TYPE_CLASS.TYPE_LINT:
			_WriteByte(TO_BYTE(Tc2_Utilities.E_ArgType.ARGTYPE_LARGE));
			_Copy(stArg.pValue, SIZEOF(LINT));

		__SYSTEM.TYPE_CLASS.TYPE_USINT:
			_WriteByte(TO_BYTE(Tc2_Utilities.E_ArgType.ARGTYPE_USINT));
			_Copy(stArg.pValue, SIZEOF(USINT));

		__SYSTEM.TYPE_CLASS.TYPE_UINT:
			_WriteByte(TO_BYTE(Tc2_Utilities.E_ArgType.ARGTYPE_UINT));
			_Copy(stArg.pValue, SIZEOF(UINT));

		__SYSTEM.TYPE_CLASS.TYPE_UDINT:
			_WriteByte(TO_BYTE(Tc2_Utilities.E_ArgType.ARGTYPE_UDINT));
			_Copy(stArg.pValue, SIZEOF(UDINT));

		__SYSTEM.TYPE_CLASS.TYPE_ULINT:
			_WriteByte(TO_BYTE(Tc2_Utilities.E_ArgType.ARGTYPE_ULARGE));
			_Copy(stArg.pValue, SIZEOF(ULINT));

		__SYSTEM.TYPE_CLASS.TYPE_REAL:
			_WriteByte(TO_BYTE(Tc2_Utilities.E_ArgType.ARGTYPE_REAL));
			_Copy(stArg.pValue, SIZEOF(REAL));

		__SYSTEM.TYPE_CLASS.TYPE_LREAL:
			_WriteByte(TO_BYTE(Tc2_Utilities.E_ArgType.ARGTYPE_LREAL));
			_Copy(stArg.pValue, SIZEOF(LREAL));

		__SYSTEM.TYPE_CLASS.TYPE_STRING:
			_WriteByte(TO_BYTE(Tc2_Utilities.E_ArgType.ARGTYPE_STRING));
			_WriteString(stArg.pValue);

		__SYSTEM.TYPE_CLASS.TYPE_WSTRING:
			_WriteByte(E_TypeIdV2.eType_WSTRING_V2);
			_WriteWString(stArg.pValue);

		__SYSTEM.TYPE_CLASS.TYPE_TIME:
			_WriteByte(E_TypeIdV2.eType_TIME_V2);
			_Copy(stArg.pValue, SIZEOF(TIME));

		__SYSTEM.TYPE_CLASS.TYPE_DATE:
			_WriteByte(E_TypeIdV2.eType_DATE_V2);
			_Copy(stArg.pValue, SIZEOF(DATE));

		__SYSTEM.TYPE_CLASS.TYPE_DATEANDTIME:
			_WriteByte(E_TypeIdV2.eType_DATE_AND_TIME_V2);
			_Copy(stArg.pValue, SIZEOF(DATE_AND_TIME));

		__SYSTEM.TYPE_CLASS.TYPE_TIMEOFDAY:
			_WriteByte(E_TypeIdV2.eType_TIME_OF_DAY_V2);
			_Copy(stArg.pValue, SIZEOF(TIME_OF_DAY));

		__SYSTEM.TYPE_CLASS.TYPE_ENUM:
			_WriteByte(E_TypeIdV2.eType_ENUM_V2);
			// Write the integer value of the enumeration
			CASE stArg.diSize OF
				1:
					_WriteByte(TO_BYTE(Tc2_Utilities.E_ArgType.ARGTYPE_BYTE));
					_Copy(stArg.pValue, SIZEOF(BYTE));
				2:
					_WriteByte(TO_BYTE(Tc2_Utilities.E_ArgType.ARGTYPE_WORD));
					_Copy(stArg.pValue, SIZEOF(WORD));
				4:
					_WriteByte(TO_BYTE(Tc2_Utilities.E_ArgType.ARGTYPE_DWORD));
					_Copy(stArg.pValue, SIZEOF(DWORD));
				8:
					_WriteByte(TO_BYTE(Tc2_Utilities.E_ArgType.ARGTYPE_LWORD));
					_Copy(stArg.pValue, SIZEOF(LWORD));
				ELSE
					_WriteByte(TO_BYTE(Tc2_Utilities.E_ArgType.ARGTYPE_UNKNOWN));
			END_CASE

		__SYSTEM.TYPE_CLASS.TYPE_LTIME:
			_WriteByte(E_TypeIdV2.eType_LTIME_V2);
			_Copy(stArg.pValue, SIZEOF(LTIME));

		ELSE
			F_InternalLog(
				E_LogLevel.eWarn,
				'FB_LogEntry.AddAnyArg',
				'Unhandled ANY type=%d',
				Tc2_Utilities.F_UDINT(stArg.TypeClass),
				Tc2_Utilities.EMPTY_ARG_VALUE,
				Tc2_Utilities.EMPTY_ARG_VALUE,
				Tc2_Utilities.EMPTY_ARG_VALUE
			);
			bError := TRUE;
	END_CASE
	nArgCount := nArgCount + 1;

ELSE
	// v1 format: existing code
	_WriteByte(1); // Type 1: Argument follows
	_WriteByte(nArgno);

	CASE stArg.TypeClass OF
		__SYSTEM.TYPE_CLASS.TYPE_BOOL:
			_WriteInt(Tc2_Utilities.E_ArgType.ARGTYPE_BOOL);
			IF Tc2_Utilities.PBYTE_TO_BYTE(stArg.pValue) <> 0 THEN
				_WriteByte(1);
			ELSE
				_WriteByte(0);
			END_IF

		__SYSTEM.TYPE_CLASS.TYPE_BYTE:
			_WriteInt(Tc2_Utilities.E_ArgType.ARGTYPE_BYTE);
			_Copy(stArg.pValue, SIZEOF(BYTE));

		__SYSTEM.TYPE_CLASS.TYPE_WORD:
			_WriteInt(Tc2_Utilities.E_ArgType.ARGTYPE_WORD);
			_Copy(stArg.pValue, SIZEOF(WORD));

		__SYSTEM.TYPE_CLASS.TYPE_DWORD:
			_WriteInt(Tc2_Utilities.E_ArgType.ARGTYPE_DWORD);
			_Copy(stArg.pValue, SIZEOF(DWORD));

		__SYSTEM.TYPE_CLASS.TYPE_LWORD:
			_WriteInt(Tc2_Utilities.E_ArgType.ARGTYPE_LWORD);
			_Copy(stArg.pValue, SIZEOF(LWORD));

		__SYSTEM.TYPE_CLASS.TYPE_SINT:
			_WriteInt(Tc2_Utilities.E_ArgType.ARGTYPE_SINT);
			_Copy(stArg.pValue, SIZEOF(SINT));

		__SYSTEM.TYPE_CLASS.TYPE_INT:
			_WriteInt(Tc2_Utilities.E_ArgType.ARGTYPE_INT);
			_Copy(stArg.pValue, SIZEOF(INT));

		__SYSTEM.TYPE_CLASS.TYPE_DINT:
			_WriteInt(Tc2_Utilities.E_ArgType.ARGTYPE_DINT);
			_Copy(stArg.pValue, SIZEOF(DINT));

		__SYSTEM.TYPE_CLASS.TYPE_LINT:
			_WriteInt(Tc2_Utilities.E_ArgType.ARGTYPE_LARGE);
			_Copy(stArg.pValue, SIZEOF(LINT));

		__SYSTEM.TYPE_CLASS.TYPE_USINT:
			_WriteInt(Tc2_Utilities.E_ArgType.ARGTYPE_USINT);
			_Copy(stArg.pValue, SIZEOF(USINT));

		__SYSTEM.TYPE_CLASS.TYPE_UINT:
			_WriteInt(Tc2_Utilities.E_ArgType.ARGTYPE_UINT);
			_Copy(stArg.pValue, SIZEOF(UINT));

		__SYSTEM.TYPE_CLASS.TYPE_UDINT:
			_WriteInt(Tc2_Utilities.E_ArgType.ARGTYPE_UDINT);
			_Copy(stArg.pValue, SIZEOF(UDINT));

		__SYSTEM.TYPE_CLASS.TYPE_ULINT:
			_WriteInt(Tc2_Utilities.E_ArgType.ARGTYPE_ULARGE);
			_Copy(stArg.pValue, SIZEOF(ULINT));

		__SYSTEM.TYPE_CLASS.TYPE_REAL:
			_WriteInt(Tc2_Utilities.E_ArgType.ARGTYPE_REAL);
			_Copy(stArg.pValue, SIZEOF(REAL));

		__SYSTEM.TYPE_CLASS.TYPE_LREAL:
			_WriteInt(Tc2_Utilities.E_ArgType.ARGTYPE_LREAL);
			_Copy(stArg.pValue, SIZEOF(LREAL));

		__SYSTEM.TYPE_CLASS.TYPE_STRING:
			_WriteInt(Tc2_Utilities.E_ArgType.ARGTYPE_STRING);
			_WriteString(stArg.pValue);

		__SYSTEM.TYPE_CLASS.TYPE_WSTRING:
			_WriteInt(E_CustomTypes.eType_WSTRING);
			_WriteWString(stArg.pValue);

		__SYSTEM.TYPE_CLASS.TYPE_TIME:
			_WriteInt(E_CustomTypes.eType_TIME);
			_Copy(stArg.pValue, SIZEOF(TIME));

		__SYSTEM.TYPE_CLASS.TYPE_DATE:
			_WriteInt(E_CustomTypes.eType_DATE);
			_Copy(stArg.pValue, SIZEOF(DATE));

		__SYSTEM.TYPE_CLASS.TYPE_DATEANDTIME:
			_WriteInt(E_CustomTypes.eType_DATE_AND_TIME);
			_Copy(stArg.pValue, SIZEOF(DATE_AND_TIME));

		__SYSTEM.TYPE_CLASS.TYPE_TIMEOFDAY:
			_WriteInt(E_CustomTypes.eType_TIME_OF_DAY);
			_Copy(stArg.pValue, SIZEOF(TIME_OF_DAY));

		__SYSTEM.TYPE_CLASS.TYPE_ENUM:
			_WriteInt(E_CustomTypes.eType_ENUM);
			// First write the integer value of the enumeration, expected 1 to 8 bytes
			CASE stArg.diSize OF
				1:
					_WriteInt(Tc2_Utilities.E_ArgType.ARGTYPE_BYTE);
					_Copy(stArg.pValue, SIZEOF(BYTE));
				2:
					_WriteInt(Tc2_Utilities.E_ArgType.ARGTYPE_WORD);
					_Copy(stArg.pValue, SIZEOF(WORD));
				4:
					_WriteInt(Tc2_Utilities.E_ArgType.ARGTYPE_DWORD);
					_Copy(stArg.pValue, SIZEOF(DWORD));
				5:
					_WriteInt(Tc2_Utilities.E_ArgType.ARGTYPE_LWORD);
					_Copy(stArg.pValue, SIZEOF(LWORD));
				ELSE
					_WriteInt(Tc2_Utilities.E_ArgType.ARGTYPE_UNKNOWN);
			END_CASE

		__SYSTEM.TYPE_CLASS.TYPE_LTIME:
			_WriteInt(E_CustomTypes.eType_LTIME);
			_Copy(stArg.pValue, SIZEOF(LTIME));

		ELSE
			F_InternalLog(
				E_LogLevel.eWarn,
				'FB_LogEntry.AddAnyArg',
				'Unhandled ANY type=%d',
				Tc2_Utilities.F_UDINT(stArg.TypeClass),
				Tc2_Utilities.EMPTY_ARG_VALUE,
				Tc2_Utilities.EMPTY_ARG_VALUE,
				Tc2_Utilities.EMPTY_ARG_VALUE
			);
			// TODO maybe rollback and ignore argument or use replacement value (null)
			bError := TRUE;
	END_CASE

END_IF

AddAnyArg := NOT bError;
END_METHOD

METHOD PUBLIC AddBuffer
VAR_INPUT
	pBuffer			: PVOID;
	nBufferLen		: UDINT;
END_VAR
_Copy(pBuffer, nBufferLen);
END_METHOD

METHOD PUBLIC AddContext
VAR_INPUT
	eScope			: E_Scope;
	pBuffer			: PVOID;
	nBufferLen		: UDINT;
END_VAR
IF bV2 THEN
	// v2 format: scope + prop_count + buffer (prop_count already included in nBufferLen)
	_WriteByte(eScope);
	_Copy(pBuffer, nBufferLen);
	nContextCount := nContextCount + 1;
ELSE
	// v1 format: existing code
	_WriteByte(2); // Type 2: Context follows
	_WriteByte(eScope);
	_Copy(pBuffer, nBufferLen);
END_IF
END_METHOD

METHOD PUBLIC AddTArg
VAR_INPUT
	nArgNo		: BYTE;
	stArg		: Tc2_Utilities.T_Arg;
END_VAR
IF bError THEN
	RETURN;
END_IF

IF stArg.eType = E_ArgType.ARGTYPE_UNKNOWN OR stArg.pData = 0 THEN
	RETURN;
END_IF

_WriteByte(1); // Type 1: Argument follows
_WriteByte(nArgNo);
_WriteInt(stArg.eType);

_Copy(ADR(stArg.eType), SIZEOF(stArg.eType));
CASE stArg.eType OF
	Tc2_Utilities.E_ArgType.ARGTYPE_BYTE:
		_Copy(stArg.pData, SIZEOF(BYTE));
	Tc2_Utilities.E_ArgType.ARGTYPE_WORD:
		_Copy(stArg.pData, SIZEOF(WORD));
	Tc2_Utilities.E_ArgType.ARGTYPE_DWORD:
		_Copy(stArg.pData, SIZEOF(DWORD));
	Tc2_Utilities.E_ArgType.ARGTYPE_REAL:
		_Copy(stArg.pData, SIZEOF(REAL));
	Tc2_Utilities.E_ArgType.ARGTYPE_LREAL:
		_Copy(stArg.pData, SIZEOF(LREAL));
	Tc2_Utilities.E_ArgType.ARGTYPE_SINT:
		_Copy(stArg.pData, SIZEOF(SINT));
	Tc2_Utilities.E_ArgType.ARGTYPE_INT:
		_Copy(stArg.pData, SIZEOF(INT));
	Tc2_Utilities.E_ArgType.ARGTYPE_DINT:
		_Copy(stArg.pData, SIZEOF(DINT));
	Tc2_Utilities.E_ArgType.ARGTYPE_USINT:
		_Copy(stArg.pData, SIZEOF(USINT));
	Tc2_Utilities.E_ArgType.ARGTYPE_UINT:
		_Copy(stArg.pData, SIZEOF(UINT));
	Tc2_Utilities.E_ArgType.ARGTYPE_UDINT:
		_Copy(stArg.pData, SIZEOF(UDINT));
	Tc2_Utilities.E_ArgType.ARGTYPE_STRING:
		_WriteString(stArg.pData);
	Tc2_Utilities.E_ArgType.ARGTYPE_BOOL:
		_WriteByte(SEL(Tc2_Utilities.PBOOL_TO_BOOL(stArg.pData), 0, 1));
	Tc2_Utilities.E_ArgType.ARGTYPE_ULARGE:
		_Copy(stArg.pData, SIZEOF(ULINT));
	Tc2_Utilities.E_ArgType.ARGTYPE_LARGE:
		_Copy(stArg.pData, SIZEOF(LINT));
	Tc2_Utilities.E_ArgType.ARGTYPE_LWORD:
		_Copy(stArg.pData, SIZEOF(LWORD));
END_CASE
END_METHOD

METHOD PUBLIC End : BOOL
VAR
	pWriteBuffer	: REFERENCE TO FB_LogBuffer;
	nBufferFree		: UINT;
	nActTaskIndex	: DINT;
	nEntryLength	: UINT;
	pEntryLenPtr	: POINTER TO UINT;
	pArgCountPtr	: POINTER TO BYTE;
	pCtxCountPtr	: POINTER TO BYTE;
END_VAR
IF bError THEN
	RETURN;
END_IF

nActTaskIndex := GETCURTASKINDEXEX();

// end buffer write access
pWriteBuffer REF= PRG_TaskLog.TaskLogger.WriteBuffer;

IF pWriteBuffer.BufferPtr <> pBuffer THEN
	// sanity check
	F_InternalLog(
		E_LogLevel.eError,
		'FB_LogEntry.End',
		'Expected buffer to be the same.',
		Tc2_Utilities.EMPTY_ARG_VALUE,
		Tc2_Utilities.EMPTY_ARG_VALUE,
		Tc2_Utilities.EMPTY_ARG_VALUE,
		Tc2_Utilities.EMPTY_ARG_VALUE
	);

	bError := TRUE;

ELSIF pWriteBuffer.BufferFree < nBufferCount THEN
	nBufferFree := TO_UINT(pWriteBuffer.BufferFree);
	F_InternalLog(
		E_LogLevel.eError,
		'FB_LogEntry.End',
		'Buffer capacity does not match buffer count. BufferFree=%d BufferCount=%d',
		Tc2_Utilities.F_UINT(nBufferFree),
		Tc2_Utilities.F_UDINT(nBufferCount),
		Tc2_Utilities.EMPTY_ARG_VALUE,
		Tc2_Utilities.EMPTY_ARG_VALUE
	);

	bError := TRUE;

ELSE
	IF bV2 THEN
		// v2: Backfill entry_length, arg_count, context_count
		// entry_length = total bytes from after the entry_length field
		nEntryLength := TO_UINT(nBufferCount - nEntryStart - 3);  // -3 for type(1) + length(2)

		// Backfill entry_length at offset
		pEntryLenPtr := pBuffer + nEntryLenOffset;
		pEntryLenPtr^ := nEntryLength;

		// Backfill arg_count at offset
		pArgCountPtr := pBuffer + nArgCountOffset;
		pArgCountPtr^ := nArgCount;

		// Backfill context_count at offset
		pCtxCountPtr := pBuffer + nCtxCountOffset;
		pCtxCountPtr^ := nContextCount;

		// No terminator for v2
		pWriteBuffer.DataAdded(nBufferCount);

		// Reset v2 flag for next use
		bV2 := FALSE;
	ELSE
		// v1: Write terminator byte
		_WriteByte(255);
		pWriteBuffer.DataAdded(nBufferCount);
	END_IF
END_IF

// Statistic
IF bError THEN
	IncUDINT(TcOtelInfo.aTaskInfo[nActTaskIndex].nAddLogToBufferErrorCount);
ELSE
	IncUDINT(TcOtelInfo.aTaskInfo[nActTaskIndex].nAddLogToBuffer);
END_IF

IF TcOtelInfo.aTaskInfo[nActTaskIndex].nMaxUsedBufferSize < pWriteBuffer.BufferUsed THEN
	TcOtelInfo.aTaskInfo[nActTaskIndex].nMaxUsedBufferSize := pWriteBuffer.BufferUsed;
END_IF

End := NOT bError;
END_METHOD

METHOD Reset
VAR_INPUT
END_VAR
_Reset();
END_METHOD

METHOD PUBLIC SetArgCount
VAR_INPUT
	nCount		: BYTE;
END_VAR
nArgCount := nCount;
END_METHOD

METHOD PUBLIC Start : BOOL
VAR_INPUT
	pLogger		: POINTER TO T_MaxString;
	pMessage		: POINTER TO T_MaxString;
	eLogLevel		: E_LogLevel;
	nTimeStampPlc	: LINT;
	nTimeStampClock	: LINT;
END_VAR
VAR
	fbSysTime		: Tc2_System.GETSYSTEMTIME;
	nTaskIndex		: DINT;
END_VAR
// Timestamp PLC
IF nTimestampPlc = 0 THEN
	fbSysTime();
	nTimeStampPlc := ULINT_TO_LINT(SHL(UDINT_TO_ULINT(fbSysTime.timeHiDW), 32) OR fbSysTime.timeLoDW);
END_IF

// Timestamp RTC
IF nTimestampClock = 0 THEN
	// F_GetActualDcTime64 reads live DC time at this instruction (LINT ns
	// since DC epoch 2000-01-01 UTC). On this runtime it advances within
	// the cycle, so each F_Log call gets a distinct ns-precise timestamp.
	// Falls back to DcTaskTime (cycle-start stamp) if DC isn't synchronised.
	nTimestampClock := TO_LINT(Tc2_EtherCAT.F_GetActualDcTime64());
	IF nTimestampClock = 0 THEN
		nTimestampClock := TwinCAT_SystemInfoVarList._TaskInfo[Tc2_System.GETCURTASKINDEXEX()].DcTaskTime;
	END_IF
END_IF

// Log-Entry Version
_WriteByte(1);

// Message
_WriteString(pMessage);

// Logger
_WriteString(pLogger);

// Level
_WriteUInt(eLogLevel);

// Timestamp PLC
_WriteLInt(nTimeStampPlc);

// Timestamp Clock
_WriteLInt(nTimeStampClock);

// Task Infos 
nTaskIndex := Tc2_System.GETCURTASKINDEXEX();
_WriteDInt(nTaskIndex);
_WriteString(ADR(TwinCAT_SystemInfoVarList._TaskInfo[nTaskIndex].TaskName));
_WriteUDInt(TwinCAT_SystemInfoVarList._TaskInfo[nTaskIndex].CycleCount);

// App Infos
_WriteString(ADR(TwinCAT_SystemInfoVarList._AppInfo.AppName));
_WriteString(ADR(TwinCAT_SystemInfoVarList._AppInfo.ProjectName));
_WriteUDInt(TwinCAT_SystemInfoVarList._AppInfo.OnlineChangeCnt);

Start := NOT bError;
END_METHOD

METHOD PUBLIC StartV2 : BOOL
VAR_INPUT
	pLogger		: POINTER TO T_MaxString;
	pMessage		: POINTER TO T_MaxString;
	eLogLevel		: E_LogLevel;
	nTimeStampPlc	: LINT;
	nTimeStampClock	: LINT;
END_VAR
VAR
	nTaskIndex		: DINT;
	stHeader		: ST_LogEntryHeaderV2;
END_VAR
// Timestamp PLC
IF nTimestampPlc = 0 THEN
	nTimeStampPlc := TO_LINT(Tc2_System.F_GetSystemTime());
END_IF

// Timestamp RTC: use DcTaskTime (cycle-accurate ns since DC epoch 2000-01-01
// UTC) instead of the ~100 ms-quantised PRG_TaskLog.RtcTime so log entries
// get the same ns-precise timestamp as push-diag samples — Grafana lines
// log rows and exceed dots up on the time axis cycle-by-cycle.
IF nTimestampClock = 0 THEN
	// F_GetActualDcTime64 reads live DC time at this instruction (LINT ns
	// since DC epoch 2000-01-01 UTC). On this runtime it advances within
	// the cycle, so each F_Log call gets a distinct ns-precise timestamp.
	// Falls back to DcTaskTime (cycle-start stamp) if DC isn't synchronised.
	nTimestampClock := TO_LINT(Tc2_EtherCAT.F_GetActualDcTime64());
	IF nTimestampClock = 0 THEN
		nTimestampClock := TwinCAT_SystemInfoVarList._TaskInfo[Tc2_System.GETCURTASKINDEXEX()].DcTaskTime;
	END_IF
END_IF

// Save entry start position for backfill calculations
nEntryStart := nBufferCount;

// Build fixed header struct (27 bytes total)
stHeader.nType := 2;						// 0x02 = v2 Log Entry
stHeader.nEntryLength := 0;					// Placeholder, backfilled in End()
stHeader.nLevel := TO_BYTE(eLogLevel);
stHeader.nTsPlc := nTimeStampPlc;			// 8 bytes
stHeader.nTsClock := nTimeStampClock;		// 8 bytes
nTaskIndex := GETCURTASKINDEXEX();
stHeader.nTaskIndex := TO_BYTE(nTaskIndex);
stHeader.nCycleCount := TwinCAT_SystemInfoVarList._TaskInfo[nTaskIndex].CycleCount;
stHeader.nArgCount := 0;					// Placeholder, backfilled in End()
stHeader.nContextCount := 0;				// Placeholder, backfilled in End()

// Save offsets for backfill
nEntryLenOffset := nBufferCount + 1;		// +1 byte for type
nArgCountOffset := nBufferCount + 25;		// type(1) + length(2) + level(1) + ts_plc(8) + ts_clock(8) + task_index(1) + cycle(4) = 25
nCtxCountOffset := nBufferCount + 26;		// nArgCount(1) after offset 25 = 26

// Write fixed header as single MEMCPY (27 bytes)
_Copy(ADR(stHeader), SIZEOF(stHeader));

// Write message string
_WriteString(pMessage);

// Write logger string (len=0 if null for default logger)
IF pLogger <> 0 THEN
	_WriteString(pLogger);
ELSE
	_WriteByte(0);	// len=0 for default logger
END_IF

// Initialize counters
nArgCount := 0;
nContextCount := 0;
bV2 := TRUE;

StartV2 := NOT bError;
END_METHOD

END_FUNCTION_BLOCK

// ---- POUs/Utils/FB_LogBuffer.TcPOU
{attribute 'no_explicit_call' := 'no direct call necessary'}
FUNCTION_BLOCK INTERNAL FB_LogBuffer
VAR
	aBuffer			: ARRAY[1..Config.nBufferLen] OF BYTE;
	nBufferCount	: UDINT;
END_VAR

PROPERTY INTERNAL BufferFree : UDINT
GET
BufferFree := Config.nBufferLen - nBufferCount;
END_GET
END_PROPERTY

PROPERTY INTERNAL BufferPtr : PVOID
GET
BufferPtr := ADR(aBuffer) + nBufferCount;
END_GET
END_PROPERTY

PROPERTY INTERNAL BufferStartPtr : PVOID
GET
BufferStartPtr := ADR(aBuffer);
END_GET
END_PROPERTY

PROPERTY INTERNAL BufferUsed : UDINT
GET
BufferUsed := nBufferCount;
END_GET
END_PROPERTY

METHOD INTERNAL Clear
nBufferCount := 0;
END_METHOD

METHOD INTERNAL DataAdded
VAR_INPUT
	nNewData		: UDINT;
END_VAR
nBufferCount := nBufferCount + nNewData;
IF nBufferCount > Config.nBufferLen THEN
	F_InternalLog(
		E_LogLevel.eError,
		'FB_LogBuffer.DataAdded',
		'Buffer overflow adding to log buffer.',
		Tc2_Utilities.EMPTY_ARG_VALUE,
		Tc2_Utilities.EMPTY_ARG_VALUE,
		Tc2_Utilities.EMPTY_ARG_VALUE,
		Tc2_Utilities.EMPTY_ARG_VALUE
	);
END_IF
END_METHOD

END_FUNCTION_BLOCK

// ---- POUs/Utils/IncUDINT.TcPOU
FUNCTION INTERNAL IncUDINT : UDINT
VAR_INPUT
	refValue		: REFERENCE TO UDINT;
END_VAR

IncUDINT := (refValue := refValue + 1);

END_FUNCTION

// ---- API/Context/F_Context.TcPOU
FUNCTION F_Context : I_ContextBuilder
VAR_STAT
	aTaskContext		: ARRAY[1..SIZEOF(TwinCAT_SystemInfoVarList._TaskInfo)/SIZEOF(PlcTaskSystemInfo)] OF FB_ContextBuilder;
END_VAR

F_Context := aTaskContext[Tc2_System.GETCURTASKINDEXEX()].Clear();

END_FUNCTION

// ---- API/Metric/FB_Metrics.TcPOU
(*
:Description: User-facing FB for capturing oversampled metric values and pushing
to tc-otel as compact batched frames.

Lifecycle pattern: declare one FB_Metrics per logical metric, ``Init`` it once
in first cycle, then call ``Observe`` with the value of any IEC scalar (or
STRING / WSTRING) you want to track. The FB:

* Locks the IEC type class on the very first ``Observe`` and rejects later
  calls of a different class — no aggregator-strategy switching mid-flight.
* Optionally rate-limits sampling (``SetSampleIntervalMs``) so a value that
  changes faster than the configured interval is sampled at most once per
  interval. Default 0 = no rate limit (every change is sampled).
* Optionally suppresses redundant samples (``SetChangeDetect``, default TRUE)
  via byte-wise comparison against the last sampled value.
* Buffers samples in an append-only body buffer (8 KB default). On overflow
  the per-frame ``flags.bit1 = ring_overflowed`` is set and additional
  samples are dropped until the next flush.
* Flushes the buffer at the configured push interval (``SetPushIntervalMs``,
  default 1000 ms). Flush also fires from ``Call()`` so users who call
  ``Observe`` only on demand still get punctual pushes.

Each frame carries header + (optional trace context) + name + unit + body.
The body is just ``sample_count * sample_size`` raw bytes — no per-sample
type/length, the receiver knows the layout from the header's ``body_schema``.

Numerics (all signed/unsigned int + REAL + LREAL) widen to LREAL (8 B). BOOL
is one byte. STRING/WSTRING are zero-padded to a per-instance fixed size
configured in ``Init``. Discrete byte-types (BYTE/WORD/DWORD/LWORD/ENUM)
are shipped raw at their native size.

**Example**

.. code-block:: pascal

    VAR
        fbMotorTemp : FB_Metrics;
    END_VAR

    IF _TaskInfo[GETCURTASKINDEXEX()].FirstCycle THEN
        fbMotorTemp.Init('motor.temperature', 'celsius');
        fbMotorTemp.SetSampleIntervalMs(100);   // at most every 100 ms
        fbMotorTemp.SetPushIntervalMs(5000);    // flush every 5 s
    END_IF

    fbMotorTemp.Observe(rTemperature);          // every cycle is fine
    PRG_TaskLog.Call();                         // pumps the per-task sender
*)
{attribute 'reflection'}
FUNCTION_BLOCK FB_Metrics
VAR_INPUT
END_VAR
VAR_OUTPUT
END_VAR
VAR CONSTANT
    (* Each frame is laid out as one contiguous byte array where the header
       grows backward into a 256-byte reserve immediately before the body.
       ADSWRITE reads a single pointer that starts at [HDR_RESERVE - hdrLen]
       and runs through the body — no MEMCPY of either region on flush.

       Header max observed size (v2 frame + 24 B trace_ctx + 63 B name + 15 B
       unit) is ~154 B; 256 B is generous padding. Body is 32 KB per half so
       a true-oversampling DC-timestamp burst (16 B / Numeric slot) fits
       ~2048 samples before mid-window autoflush kicks in. Total per-half =
       HDR_RESERVE + BODY_CAPACITY = 33024 B.

       Autoflush high-water mark: when _nBodyOffset crosses 4/5 of
       BODY_CAPACITY the next append triggers _DoFlush, swapping halves
       mid-window so the burst keeps streaming. *)
    HDR_RESERVE             : UDINT := 256;
    BODY_CAPACITY           : UDINT := 32768;
    BODY_HIGH_WATER         : UDINT := 26214;         // BODY_CAPACITY * 4 / 5
    FRAME_SIZE              : UDINT := 33024;         // HDR_RESERVE + BODY_CAPACITY
END_VAR
VAR
    (* Identification *)
    _bInitialized       : BOOL;
    _sName              : STRING(63);
    _sUnit              : STRING(15);
    _nMetricId          : UDINT;                      // FNV-1a(name)

    (* Type lock — set on first Observe *)
    _eBodySchema        : E_MetricBodySchema;         // eUnknown until first Observe
    _nSampleSize        : UDINT;                      // bytes per sample in body
    _nLockedTypeClass   : __SYSTEM.TYPE_CLASS;
    _nStringSize        : UDINT := 64;                // for eString / eWstring; bytes for eString, chars for eWstring

    (* Phase 8 — A/B frame layout. Each half is one contiguous byte array
       with the header staged into [HDR_RESERVE - hdrLen .. HDR_RESERVE - 1]
       and body samples appended from [HDR_RESERVE..]. Observe writes into
       whichever half is ACTIVE; the pending half stays frozen while the
       sender ships it via ADSWRITE with SRCADDR pointing directly here.
       No MEMCPY of the body on flush. *)
    _aFrameA            : ARRAY[0..33023] OF BYTE;
    _aFrameB            : ARRAY[0..33023] OF BYTE;
    _eActiveBuf         : USINT;                      // 0 = A is active, 1 = B is active

    (* Active-half mutable state. Reset on flush when the active half flips. *)
    _nBodyOffset        : UDINT;                      // bytes appended into active body region (from HDR_RESERVE)
    _nSampleCount       : UDINT;
    _bOverflow          : BOOL;

    (* Pending-half snapshot — owned by the sender from Enqueue until the
       _NotifyFrameSent callback. Stable pointer region:
       frame[HDR_RESERVE - _nPendingHdrLen .. HDR_RESERVE + _nPendingBodyLen - 1]. *)
    _bPending           : BOOL;
    _ePendingBuf        : USINT;                      // 0 = A is pending, 1 = B is pending
    _nPendingHdrLen     : UDINT;
    _nPendingBodyLen    : UDINT;

    (* Change-detect cache — first 64 B of the last sampled value. Long
       strings (>64 B) lose change-detect precision past byte 64; this
       is acceptable for typical state strings. *)
    _abyLastValue       : ARRAY[0..63] OF BYTE;
    _bLastValueValid    : BOOL;
    _bChangeDetect      : BOOL := TRUE;

    (* Timing — uses task cycle counter converted to cycle targets so it
       agrees with FB_TcOtelTaskDiag and survives RtcTime jitter / sync. *)
    _nSampleIntervalMs  : UDINT;                      // 0 = no rate limit
    _nPushIntervalMs    : UDINT := 1000;
    _nLastSampleCycle   : UDINT;
    _bLastSampleSet     : BOOL;
    _nWindowStartCycle  : UDINT;
    _bWindowStartSet    : BOOL;

    (* Window content *)
    _nCycleStart        : UDINT;
    _nCycleEnd          : UDINT;
    _nDcTimeStart       : LINT;
    _nDcTimeEnd         : LINT;
    _bWindowHasSample   : BOOL;

    (* Counters surfaced for online inspection *)
    _nFlushOk           : UDINT;
    _nDropAppend        : UDINT;                      // appends dropped (active body overflow)
    _nDropEmit          : UDINT;                      // sender ring full / ADSWRITE err
    _nDropWindow        : UDINT;                      // window expired while previous still queued
    _nWrongTypeDrops    : UDINT;                      // Observe called with type ≠ locked

    (* Phase 7 — bitmask aggregation. When _nStatMask > 0 and the locked
       schema is numeric, Observe updates the aggregator on every call
       (Welford online for mean/stddev) instead of just rate-limiting.
       At each sample tick popcount(_nStatMask) LREALs are written into
       the body in bit-order (Min, Max, Mean, Sum, Count, StdDev) and the
       aggregator resets. Mask=0 keeps the original raw-sample behaviour. *)
    _nStatMask          : BYTE;                       // E_MetricStat bitmask, 0 = raw
    _nAggSampleSize     : UDINT;                      // popcount(mask) * 8, cached
    _aggMin             : LREAL;
    _aggMax             : LREAL;
    _aggMean            : LREAL;                      // Welford running mean
    _aggSumSq           : LREAL;                      // sum of squared deltas (Welford M2)
    _aggSum             : LREAL;
    _nAggCount          : UDINT;
    _bAggHasSample      : BOOL;                       // first observation in current window seen?

    (* Trace-context binding (Phase 5).
       _pTracer is set persistently by BindTracer — at flush time the
       tracer's innermost open span is snapshotted into the frame.
       _pSpanOverride is set by WithSpan and consumed by the very next
       flush — lets users force a specific span when "innermost" isn't
       what they want. *)
    _pTracer            : REFERENCE TO FB_Trace;
    _pSpanOverride      : REFERENCE TO FB_Span;

    (* Per-sample timestamps (opt-in). When TRUE each body slot is prefixed
       with a 2-byte little-endian u16 cycle offset (relative to
       _nCycleStart). _CheckFlush caps the push window at 0xFFFF cycles to
       keep u16 safe; receiver-side decoders gate on the matching header flag
       METRIC_FLAG_HAS_SAMPLE_TS (0x04). *)
    _bRecordSampleTimes   : BOOL;

    (* High-resolution per-sample timestamps for true oversampling. When TRUE
       each body slot is prefixed with an 8-byte little-endian i64 absolute
       DC time — the raw F_GetActualDcTime64() reading at the Observe call.
       Mutually exclusive with _bRecordSampleTimes; setting both is a
       programming error. Receiver-side decoders gate on the matching header
       flag METRIC_FLAG_HAS_SAMPLE_TS_DC (0x10). Slot stride becomes
       _nSampleSize + 8. No tiebreaker — duplicate DC reads inside one task
       cycle stay duplicate so emitted timestamps don't lie about the
       hardware clock. *)
    _bRecordSampleTimesDc : BOOL;

    (* Phase 2 scope-resolver: instance path of the owning FB.
       FB_Init strips the library + application + variable-name
       segments, leaving (e.g.) ``PRG_Foo.fbBar`` in ``_sLogger``.
       Emitted as the trailing namespace string on the metric
       aggregate frame when non-empty; tc-otel's ScopeResolver
       maps it to the owning FB's TYPE for ``scope.name``. *)
    {attribute 'instance-path'}
    {attribute 'noinit'}
    _sInstancePath      : T_MaxString;
    _sLogger            : T_MaxString;
END_VAR

(*
:Description: Byte pointer to the start of the body region in the ACTIVE frame.

Body writes land at ``_ActiveBodyPtr() + _nBodyOffset``. Swapping buffers
at flush time only toggles ``_eActiveBuf``; subsequent Observe calls land
in the now-fresh half without touching the pending half still being shipped.
*)
METHOD PRIVATE _ActiveBodyPtr : POINTER TO BYTE
IF _eActiveBuf = 0 THEN
    _ActiveBodyPtr := ADR(_aFrameA[HDR_RESERVE]);
ELSE
    _ActiveBodyPtr := ADR(_aFrameB[HDR_RESERVE]);
END_IF
END_METHOD

(*
:Description: Byte pointer to the start of the ACTIVE frame (i.e. the header
reserve base). Used by _DoFlush to position the header immediately before the
body via ``_ActiveFrameAddr() + (HDR_RESERVE - hdrLen)``.
*)
METHOD PRIVATE _ActiveFrameAddr : POINTER TO BYTE
IF _eActiveBuf = 0 THEN
    _ActiveFrameAddr := ADR(_aFrameA[0]);
ELSE
    _ActiveFrameAddr := ADR(_aFrameB[0]);
END_IF
END_METHOD

(*
:Description: Clear the Welford aggregator state at the start of every sample window.
*)
METHOD PRIVATE _AggReset
_aggMin        := 0.0;
_aggMax        := 0.0;
_aggMean       := 0.0;
_aggSumSq      := 0.0;
_aggSum        := 0.0;
_nAggCount     := 0;
_bAggHasSample := FALSE;
END_METHOD

(*
:Description: Fold one observation into the Welford online aggregator.

Maintains running min/max/sum/count exactly, and mean / sum-of-squared-
deltas via Welford so the per-Observe cost stays at ~6 LREAL ops without
ever rebuilding from a stored sample list. StdDev is derived from
``_aggSumSq / (n - 1)`` only at flush time.

Reference: B. P. Welford, *Note on a Method for Calculating Corrected
Sums of Squares and Products*, Technometrics 4(3), 1962.
*)
METHOD PRIVATE _AggUpdate
VAR_INPUT
    fValue : LREAL;
END_VAR
VAR
    fDelta  : LREAL;
    fDelta2 : LREAL;
END_VAR
IF NOT _bAggHasSample THEN
    _aggMin        := fValue;
    _aggMax        := fValue;
    _aggMean       := fValue;
    _aggSumSq      := 0.0;
    _aggSum        := fValue;
    _nAggCount     := 1;
    _bAggHasSample := TRUE;
ELSE
    IF fValue < _aggMin THEN
        _aggMin := fValue;
    END_IF
    IF fValue > _aggMax THEN
        _aggMax := fValue;
    END_IF
    _aggSum    := _aggSum + fValue;
    _nAggCount := _nAggCount + 1;
    fDelta     := fValue - _aggMean;
    _aggMean   := _aggMean + fDelta / UDINT_TO_LREAL(_nAggCount);
    fDelta2    := fValue - _aggMean;
    _aggSumSq  := _aggSumSq + fDelta * fDelta2;
END_IF
END_METHOD

(*
:Description: Widen any IEC numeric (or BOOL) to LREAL.

